C01735=-85.269,-50.626,61.037,-179.1730,-2.3238,-10409.3015
C01736=-88.593,-46.265,61.359,-179.9976,-0.1564,-10412.4256
C01737=-91.197,-41.009,61.571,179.9982,-0.0180,-10415.7877
C01738=-93.484,-35.488,61.571,179.9993,-0.0181,-10419.2124
C01739=-95.359,-29.931,61.359,179.9991,-0.1559,-10422.5741
C01740=-96.092,-24.496,61.037,179.1715,-2.3205,-10425.6986
C01741=-94.474,-19.672,60.719,176.6107,-3.5414,-10428.2376
C01742=-90.884,-16.396,60.330,172.2930,-2.2395,-10429.7735
C01743=-85.905,-15.041,59.597,172.0939,-0.5331,-10430.0688
C01744=-80.549,-13.963,58.128,174.0620,-0.3468,-10430.1656
C01745=-75.822,-12.951,56.240,177.3643,-0.2478,-10430.3070
C01746=-72.328,-11.825,54.436,-175.3679,1.0293,-10430.7148
C01747=-70.362,-9.959,53.146,-160.4056,25.5283,-10431.9439
C01748=-69.984,-6.412,52.637,-175.1539,38.4339,-10434.7651
C01749=-70.158,-3.072,52.615,179.7154,39.0245,-10437.4928
C01750=-70.224,0.000,52.630,180.0000,39.0133,-10440.0000
C01751=-70.158,3.071,52.615,-179.7148,39.0245,-10442.5064
C01752=-69.984,6.412,52.637,175.1539,38.4339,-10445.2349
C01753=-70.362,9.959,53.146,160.4106,25.5345,-10448.0561
C01754=-72.328,11.825,54.436,175.3679,1.0293,-10449.2852
C01755=-75.822,12.951,56.240,-177.3643,-0.2478,-10449.6930
C01756=-80.549,13.963,58.128,-174.0620,-0.3468,-10449.8344
C01757=-85.905,15.041,59.597,-172.0939,-0.5331,-10449.9312
C01758=-90.884,16.396,60.330,-172.2930,-2.2395,-10450.2265
C01759=-94.474,19.672,60.719,-176.6107,-3.5414,-10451.7624
C01760=-96.092,24.496,61.037,-179.1715,-2.3205,-10454.3014
C01761=-95.359,29.931,61.359,-179.9991,-0.1559,-10457.4259
C01762=-93.484,35.488,61.571,-179.9993,-0.0181,-10460.7876
C01763=-91.197,41.009,61.571,-179.9982,-0.0180,-10464.2123
C01764=-88.593,46.265,61.359,179.9976,-0.1564,-10467.5744
C01765=-85.269,50.626,61.037,179.1730,-2.3238,-10470.6985
C01766=-80.714,52.893,60.719,176.6123,-3.5381,-10473.2374
C01767=-75.858,52.671,60.330,172.2916,-2.2418,-10474.7737
C01768=-71.379,50.109,59.597,172.0924,-0.5334,-10475.0694
C01769=-66.830,47.084,58.128,174.0623,-0.3437,-10475.1660
C01770=-62.772,44.457,56.240,177.3670,-0.2495,-10475.3073
C01771=-59.505,42.782,54.436,-175.3684,1.0288,-10475.7148
C01772=-56.796,42.712,53.146,-160.4096,25.5319,-10476.9441
C01773=-54.020,44.952,52.637,-175.1533,38.4356,-10479.7651
C01774=-51.781,47.437,52.615,179.7155,39.0245,-10482.4931
C01775=-49.656,49.656,52.630,179.9948,39.0149,-10485.0000
C01776=-47.437,51.781,52.615,-179.7155,39.0245,-10487.5069
C01777=-44.952,54.020,52.637,175.1533,38.4356,-10490.2349
C01778=-42.711,56.796,53.146,160.4094,25.5317,-10493.0566
C01779=-42.782,59.505,54.436,175.3684,1.0288,-10494.2852
C01780=-44.457,62.772,56.240,-177.3670,-0.2495,-10494.6927
C01781=-47.084,66.830,58.128,-174.0623,-0.3437,-10494.8340
C01782=-50.109,71.379,59.597,-172.0924,-0.5334,-10494.9306
C01783=-52.671,75.858,60.330,-172.2916,-2.2418,-10495.2263
C01784=-52.893,80.714,60.719,-176.6123,-3.5381,-10496.7626
C01785=-50.626,85.269,61.037,-179.1730,-2.3238,-10499.3015
C01786=-46.265,88.593,61.359,-179.9976,-0.1564,-10502.4256
C01787=-41.009,91.197,61.571,179.9982,-0.0180,-10505.7877
C01788=-35.488,93.484,61.571,179.9993,-0.0181,-10509.2124
C01789=-29.931,95.359,61.359,179.9991,-0.1559,-10512.5741
C01790=-24.496,96.092,61.037,179.1715,-2.3205,-10515.6986
C01791=-19.672,94.474,60.719,176.6107,-3.5414,-10518.2376
C01792=-16.396,90.884,60.330,172.2930,-2.2395,-10519.7735
C01793=-15.041,85.905,59.597,172.0939,-0.5331,-10520.0688
C01794=-13.963,80.549,58.128,174.0620,-0.3468,-10520.1656
C01795=-12.951,75.822,56.240,177.3643,-0.2478,-10520.3070
C01796=-11.825,72.328,54.436,-175.3679,1.0293,-10520.7148
C01797=-9.959,70.362,53.146,-160.4106,25.5345,-10521.9439
C01798=-6.412,69.984,52.637,-175.1539,38.4339,-10524.7651
C01799=-3.071,70.158,52.615,179.7148,39.0245,-10527.4936
C01800=0.000,68.843,54.342,-180.0000,38.7770,-10530.0000
C01801=2.945,68.781,54.326,-179.7056,38.7871,-10532.4517
C01802=6.200,68.619,54.350,174.8933,38.1355,-10535.1629
C01803=9.699,69.044,54.888,160.3569,24.2302,-10537.9963
C01804=11.507,71.127,56.252,176.4195,0.6994,-10539.1897
C01805=12.586,74.809,58.158,-176.9112,-0.2537,-10539.5501
C01806=13.569,79.780,60.151,-173.8939,-0.2961,-10539.6525
C01807=14.621,85.405,61.698,-172.0565,-0.4508,-10539.7146
C01808=15.942,90.636,62.469,-172.2266,-2.1131,-10539.9757
C01809=19.246,94.423,62.877,-176.5198,-3.5287,-10541.5206
C01810=24.159,96.154,63.210,-179.1544,-2.3288,-10544.1038
C01811=29.718,95.429,63.547,-179.9995,-0.1559,-10547.2974
C01812=35.416,93.512,63.770,-179.9993,-0.0181,-10550.7433
C01813=41.080,91.166,63.770,-179.9982,-0.0180,-10554.2566
C01814=46.465,88.493,63.547,179.9980,-0.1564,-10557.7026
C01815=50.908,85.074,63.210,179.1554,-2.3286,-10560.8962
C01816=53.158,80.376,62.877,176.5237,-3.5316,-10563.4793
C01817=52.817,75.362,62.469,172.2314,-2.1139,-10565.0245
C01818=50.052,70.729,61.698,172.0558,-0.4490,-10565.2855
C01819=46.818,66.007,60.151,173.8890,-0.2958,-10565.3476
C01820=43.998,61.798,58.158,176.9122,-0.2494,-10565.4495
C01821=42.158,58.431,56.252,-176.4248,0.6998,-10565.8105
C01822=41.963,55.679,54.888,-160.3550,24.2338,-10567.0038
C01823=44.137,52.905,54.350,-174.8913,38.1376,-10569.8372
C01824=46.553,50.718,54.326,179.7087,38.7878,-10572.5482
C01825=48.679,48.679,54.342,179.9948,38.7763,-10575.0000
C01826=50.718,46.553,54.326,-179.7087,38.7878,-10577.4518
C01827=52.905,44.137,54.350,174.8913,38.1376,-10580.1628
C01828=55.680,41.963,54.888,160.3548,24.2336,-10582.9966
C01829=58.431,42.158,56.252,176.4248,0.6998,-10584.1895
C01830=61.798,43.998,58.158,-176.9122,-0.2494,-10584.5505
C01831=66.007,46.818,60.151,-173.8890,-0.2958,-10584.6524
C01832=70.729,50.052,61.698,-172.0558,-0.4490,-10584.7145
C01833=75.362,52.817,62.469,-172.2314,-2.1139,-10584.9755
C01834=80.376,53.158,62.877,-176.5237,-3.5316,-10586.5207
C01835=85.074,50.908,63.210,-179.1554,-2.3286,-10589.1038
C01836=88.493,46.465,63.547,-179.9980,-0.1564,-10592.2974
C01837=91.166,41.080,63.770,179.9982,-0.0180,-10595.7434
C01838=93.512,35.416,63.770,179.9993,-0.0181,-10599.2567
C01839=95.429,29.718,63.547,179.9995,-0.1559,-10602.7026
C01840=96.154,24.159,63.210,179.1544,-2.3288,-10605.8962
C01841=94.423,19.246,62.877,176.5198,-3.5287,-10608.4794
C01842=90.636,15.942,62.469,172.2266,-2.1131,-10610.0243
C01843=85.405,14.621,61.698,172.0565,-0.4508,-10610.2854
C01844=79.780,13.569,60.151,173.8939,-0.2961,-10610.3475
C01845=74.809,12.586,58.158,176.9112,-0.2537,-10610.4499
C01846=71.127,11.507,56.252,-176.4195,0.6994,-10610.8103
C01847=69.044,9.699,54.888,-160.3569,24.2302,-10612.0037
C01848=68.619,6.200,54.350,-174.8933,38.1355,-10614.8371
C01849=68.781,2.945,54.326,179.7056,38.7871,-10617.5483
C01850=68.843,0.000,54.342,-180.0000,38.7770,-10620.0000
C01851=68.781,-2.945,54.326,-179.7056,38.7871,-10622.4517
C01852=68.619,-6.200,54.350,174.8933,38.1355,-10625.1629
C01853=69.044,-9.699,54.888,160.3561,24.2357,-10627.9963
C01854=71.127,-11.507,56.252,176.4195,0.6994,-10629.1897
C01855=74.809,-12.586,58.158,-176.9112,-0.2537,-10629.5501
C01856=79.780,-13.569,60.151,-173.8939,-0.2961,-10629.6525
C01857=85.405,-14.621,61.698,-172.0565,-0.4508,-10629.7146
C01858=90.636,-15.942,62.469,-172.2266,-2.1131,-10629.9757
C01859=94.423,-19.246,62.877,-176.5198,-3.5287,-10631.5206
C01860=96.154,-24.159,63.210,-179.1544,-2.3288,-10634.1038
C01861=95.429,-29.718,63.547,-179.9995,-0.1559,-10637.2974
C01862=93.512,-35.416,63.770,-179.9993,-0.0181,-10640.7433
C01863=91.166,-41.080,63.770,-179.9982,-0.0180,-10644.2566
C01864=88.493,-46.465,63.547,179.9980,-0.1564,-10647.7026
C01865=85.074,-50.908,63.210,179.1554,-2.3286,-10650.8962
C01866=80.376,-53.158,62.877,176.5237,-3.5316,-10653.4793
C01867=75.362,-52.817,62.469,172.2314,-2.1139,-10655.0245
C01868=70.729,-50.052,61.698,172.0558,-0.4490,-10655.2855
C01869=66.007,-46.818,60.151,173.8890,-0.2958,-10655.3476
C01870=61.798,-43.998,58.158,176.9122,-0.2494,-10655.4495
C01871=58.431,-42.158,56.252,-176.4248,0.6998,-10655.8105
C01872=55.679,-41.963,54.888,-160.3550,24.2338,-10657.0038
C01873=52.905,-44.137,54.350,-174.8913,38.1376,-10659.8372
C01874=50.718,-46.553,54.326,179.7087,38.7878,-10662.5482
C01875=48.679,-48.679,54.342,179.9948,38.7763,-10665.0000
C01876=46.553,-50.718,54.326,-179.7087,38.7878,-10667.4518
C01877=44.137,-52.905,54.350,174.8913,38.1376,-10670.1628
C01878=41.963,-55.680,54.888,160.3548,24.2336,-10672.9966
C01879=42.158,-58.431,56.252,176.4248,0.6998,-10674.1895
C01880=43.998,-61.798,58.158,-176.9122,-0.2494,-10674.5505
C01881=46.818,-66.007,60.151,-173.8890,-0.2958,-10674.6524
C01882=50.052,-70.729,61.698,-172.0558,-0.4490,-10674.7145
C01883=52.817,-75.362,62.469,-172.2314,-2.1139,-10674.9755
C01884=53.158,-80.376,62.877,-176.5237,-3.5316,-10676.5207
C01885=50.908,-85.074,63.210,-179.1554,-2.3286,-10679.1038
C01886=46.465,-88.493,63.547,-179.9980,-0.1564,-10682.2974
C01887=41.080,-91.166,63.770,179.9982,-0.0180,-10685.7434
C01888=35.416,-93.512,63.770,179.9993,-0.0181,-10689.2567
C01889=29.718,-95.429,63.547,179.9995,-0.1559,-10692.7026
C01890=24.159,-96.154,63.210,179.1544,-2.3288,-10695.8962
C01891=19.246,-94.423,62.877,176.5198,-3.5287,-10698.4794
C01892=15.942,-90.636,62.469,172.2266,-2.1131,-10700.0243
C01893=14.621,-85.405,61.698,172.0565,-0.4508,-10700.2854
C01894=13.569,-79.780,60.151,173.8939,-0.2961,-10700.3475
C01895=12.586,-74.809,58.158,176.9112,-0.2537,-10700.4499
C01896=11.507,-71.127,56.252,-176.4195,0.6994,-10700.8103
C01897=9.699,-69.044,54.888,-160.3569,24.2302,-10702.0037
C01898=6.200,-68.619,54.350,-174.8933,38.1355,-10704.8371
C01899=2.945,-68.781,54.326,179.7056,38.7871,-10707.5483
C01900=0.000,-68.843,54.342,-180.0000,38.7770,-10710.0000
C01901=-2.945,-68.781,54.326,-179.7056,38.7871,-10712.4517
C01902=-6.200,-68.619,54.350,174.8933,38.1355,-10715.1629
C01903=-9.699,-69.044,54.888,160.3561,24.2357,-10717.9963
C01904=-11.507,-71.127,56.252,176.4195,0.6994,-10719.1897
C01905=-12.586,-74.809,58.158,-176.9112,-0.2537,-10719.5501
C01906=-13.569,-79.780,60.151,-173.8939,-0.2961,-10719.6525
C01907=-14.621,-85.405,61.698,-172.0565,-0.4508,-10719.7146
C01908=-15.942,-90.636,62.469,-172.2266,-2.1131,-10719.9757
C01909=-19.246,-94.423,62.877,-176.5198,-3.5287,-10721.5206
C01910=-24.159,-96.154,63.210,-179.1544,-2.3288,-10724.1038
C01911=-29.718,-95.429,63.547,-179.9995,-0.1559,-10727.2974
C01912=-35.416,-93.512,63.770,-179.9993,-0.0181,-10730.7433
C01913=-41.080,-91.166,63.770,-179.9982,-0.0180,-10734.2566
C01914=-46.465,-88.493,63.547,179.9980,-0.1564,-10737.7026
C01915=-50.908,-85.074,63.210,179.1554,-2.3286,-10740.8962
C01916=-53.158,-80.376,62.877,176.5237,-3.5316,-10743.4793
C01917=-52.817,-75.362,62.469,172.2314,-2.1139,-10745.0245
C01918=-50.052,-70.729,61.698,172.0558,-0.4490,-10745.2855
C01919=-46.818,-66.007,60.151,173.8890,-0.2958,-10745.3476
C01920=-43.998,-61.798,58.158,176.9122,-0.2494,-10745.4495
C01921=-42.158,-58.431,56.252,-176.4248,0.6998,-10745.8105
C01922=-41.963,-55.679,54.888,-160.3550,24.2338,-10747.0038
C01923=-44.137,-52.905,54.350,-174.8913,38.1376,-10749.8372
C01924=-46.553,-50.718,54.326,179.7087,38.7878,-10752.5482
C01925=-48.679,-48.679,54.342,179.9948,38.7763,-10755.0000
C01926=-50.718,-46.553,54.326,-179.7087,38.7878,-10757.4518
C01927=-52.905,-44.137,54.350,174.8913,38.1376,-10760.1628
C01928=-55.680,-41.963,54.888,160.3548,24.2336,-10762.9966
C01929=-58.431,-42.158,56.252,176.4248,0.6998,-10764.1895
C01930=-61.798,-43.998,58.158,-176.9122,-0.2494,-10764.5505
C01931=-66.007,-46.818,60.151,-173.8890,-0.2958,-10764.6524
C01932=-70.729,-50.052,61.698,-172.0558,-0.4490,-10764.7145
C01933=-75.362,-52.817,62.469,-172.2314,-2.1139,-10764.9755
C01934=-80.376,-53.158,62.877,-176.5237,-3.5316,-10766.5207
C01935=-85.074,-50.908,63.210,-179.1554,-2.3286,-10769.1038
C01936=-88.493,-46.465,63.547,-179.9980,-0.1564,-10772.2974
C01937=-91.166,-41.080,63.770,179.9982,-0.0180,-10775.7434
C01938=-93.512,-35.416,63.770,179.9993,-0.0181,-10779.2567
C01939=-95.429,-29.718,63.547,179.9995,-0.1559,-10782.7026
C01940=-96.154,-24.159,63.210,179.1544,-2.3288,-10785.8962
C01941=-94.423,-19.246,62.877,176.5198,-3.5287,-10788.4794
C01942=-90.636,-15.942,62.469,172.2266,-2.1131,-10790.0243
C01943=-85.405,-14.621,61.698,172.0565,-0.4508,-10790.2854
C01944=-79.780,-13.569,60.151,173.8939,-0.2961,-10790.3475
C01945=-74.809,-12.586,58.158,176.9112,-0.2537,-10790.4499
C01946=-71.127,-11.507,56.252,-176.4195,0.6994,-10790.8103
C01947=-69.044,-9.699,54.888,-160.3569,24.2302,-10792.0037
C01948=-68.619,-6.200,54.350,-174.8933,38.1355,-10794.8371
C01949=-68.781,-2.945,54.326,179.7056,38.7871,-10797.5483
C01950=-68.843,0.000,54.342,180.0000,38.7770,-10800.0000
C01951=-68.781,2.945,54.326,-179.7056,38.7871,-10802.4517
C01952=-68.619,6.200,54.350,174.8933,38.1355,-10805.1629
C01953=-69.044,9.699,54.888,160.3561,24.2357,-10807.9963
C01954=-71.127,11.507,56.252,176.4195,0.6994,-10809.1897
C01955=-74.809,12.586,58.158,-176.9112,-0.2537,-10809.5501
C01956=-79.780,13.569,60.151,-173.8939,-0.2961,-10809.6525
C01957=-85.405,14.621,61.698,-172.0565,-0.4508,-10809.7146
C01958=-90.636,15.942,62.469,-172.2266,-2.1131,-10809.9757
C01959=-94.423,19.246,62.877,-176.5198,-3.5287,-10811.5206
C01960=-96.154,24.159,63.210,-179.1544,-2.3288,-10814.1038
C01961=-95.429,29.718,63.547,-179.9995,-0.1559,-10817.2974
C01962=-93.512,35.416,63.770,-179.9993,-0.0181,-10820.7433
C01963=-91.166,41.080,63.770,-179.9982,-0.0180,-10824.2566
C01964=-88.493,46.465,63.547,179.9980,-0.1564,-10827.7026
C01965=-85.074,50.908,63.210,179.1554,-2.3286,-10830.8962
C01966=-80.376,53.158,62.877,176.5237,-3.5316,-10833.4793
C01967=-75.362,52.817,62.469,172.2314,-2.1139,-10835.0245
C01968=-70.729,50.052,61.698,172.0558,-0.4490,-10835.2855
C01969=-66.007,46.818,60.151,173.8890,-0.2958,-10835.3476
C01970=-61.798,43.998,58.158,176.9122,-0.2494,-10835.4495
C01971=-58.431,42.158,56.252,-176.4248,0.6998,-10835.8105
C01972=-55.679,41.963,54.888,-160.3550,24.2338,-10837.0038
C01973=-52.905,44.137,54.350,-174.8913,38.1376,-10839.8372
C01974=-50.718,46.553,54.326,179.7087,38.7878,-10842.5482
C01975=-48.679,48.679,54.342,179.9948,38.7763,-10845.0000
C01976=-46.553,50.718,54.326,-179.7087,38.7878,-10847.4518
C01977=-44.137,52.905,54.350,174.8913,38.1376,-10850.1628
C01978=-41.963,55.680,54.888,160.3548,24.2336,-10852.9966
C01979=-42.158,58.431,56.252,176.4248,0.6998,-10854.1895
C01980=-43.998,61.798,58.158,-176.9122,-0.2494,-10854.5505
C01981=-46.818,66.007,60.151,-173.8890,-0.2958,-10854.6524
C01982=-50.052,70.729,61.698,-172.0558,-0.4490,-10854.7145
C01983=-52.817,75.362,62.469,-172.2314,-2.1139,-10854.9755
C01984=-53.158,80.376,62.877,-176.5237,-3.5316,-10856.5207
C01985=-50.908,85.074,63.210,-179.1554,-2.3286,-10859.1038
C01986=-46.465,88.493,63.547,-179.9980,-0.1564,-10862.2974
C01987=-41.080,91.166,63.770,179.9982,-0.0180,-10865.7434
C01988=-35.416,93.512,63.770,179.9993,-0.0181,-10869.2567
C01989=-29.718,95.429,63.547,179.9995,-0.1559,-10872.7026
C01990=-24.159,96.154,63.210,179.1544,-2.3288,-10875.8962
C01991=-19.246,94.423,62.877,176.5198,-3.5287,-10878.4794
C01992=-15.942,90.636,62.469,172.2266,-2.1131,-10880.0243
C01993=-14.621,85.405,61.698,172.0565,-0.4508,-10880.2854
C01994=-13.569,79.780,60.151,173.8939,-0.2961,-10880.3475
C01995=-12.586,74.809,58.158,176.9112,-0.2537,-10880.4499
C01996=-11.507,71.127,56.252,-176.4195,0.6994,-10880.8103
C01997=-9.699,69.044,54.888,-160.3561,24.2357,-10882.0037
C01998=-6.200,68.619,54.350,-174.8933,38.1355,-10884.8371
C01999=-2.945,68.781,54.326,179.7056,38.7871,-10887.5483
///TOOL 0
///POSTYPE ANGLE
///ANGLE
EC00000=38.2428,7290.0000
EC00001=38.2510,7292.8792
EC00002=38.0004,7295.7259
EC00003=32.4399,7298.4654
EC00004=8.6017,7299.9566
EC00005=1.1820,7300.7254
EC00006=-0.3684,7301.2119
EC00007=-1.1362,7301.6495
EC00008=-2.4170,7302.2909
EC00009=-2.2669,7303.8024
EC00010=-1.5763,7305.9922
EC00011=-0.0779,7308.5312
EC00012=-0.0128,7311.1696
EC00013=-0.0128,7313.8303
EC00014=-0.0769,7316.4689
EC00015=-1.5754,7319.0082
EC00016=-2.2635,7321.1977
EC00017=-2.4130,7322.7089
EC00018=-1.1367,7323.3509
EC00019=-0.3687,7323.7878
EC00020=1.1799,7324.2746
EC00021=8.5989,7325.0436
EC00022=32.4425,7326.5348
EC00023=38.0014,7329.2737
EC00024=38.2519,7332.1206
EC00025=38.2429,7335.0000
EC00026=38.2519,7337.8789
EC00027=38.0014,7340.7263
EC00028=32.4425,7343.4652
EC00029=8.5989,7344.9564
EC00030=1.1799,7345.7254
EC00031=-0.3687,7346.2122
EC00032=-1.1367,7346.6491
EC00033=-2.4130,7347.2911
EC00034=-2.2635,7348.8023
EC00035=-1.5754,7350.9918
EC00036=-0.0769,7353.5311
EC00037=-0.0128,7356.1697
EC00038=-0.0128,7358.8304
EC00039=-0.0779,7361.4688
EC00040=-1.5763,7364.0078
EC00041=-2.2669,7366.1976
EC00042=-2.4170,7367.7091
EC00043=-1.1362,7368.3505
EC00044=-0.3684,7368.7881
EC00045=1.1820,7369.2746
EC00046=8.6017,7370.0434
EC00047=32.4399,7371.5346
EC00048=38.0004,7374.2741
EC00049=38.2510,7377.1208
EC00050=38.2428,7380.0000
EC00051=38.2510,7382.8792
EC00052=38.0004,7385.7266
EC00053=32.4399,7388.4654
EC00054=8.6017,7389.9566
EC00055=1.1820,7390.7254
EC00056=-0.3684,7391.2119
EC00057=-1.1362,7391.6495
EC00058=-2.4170,7392.2909
EC00059=-2.2669,7393.8024
EC00060=-1.5763,7395.9922
EC00061=-0.0779,7398.5312
EC00062=-0.0128,7401.1696
EC00063=-0.0128,7403.8303
EC00064=-0.0769,7406.4689
EC00065=-1.5754,7409.0082
EC00066=-2.2635,7411.1977
EC00067=-2.4130,7412.7089
EC00068=-1.1367,7413.3509
EC00069=-0.3687,7413.7878
EC00070=1.1799,7414.2746
EC00071=8.5989,7415.0436
EC00072=32.4425,7416.5348
EC00073=38.0014,7419.2737
EC00074=38.2519,7422.1206
EC00075=38.2429,7425.0000
EC00076=38.2519,7427.8789
EC00077=38.0014,7430.7263
EC00078=32.4425,7433.4652
EC00079=8.5989,7434.9564
EC00080=1.1799,7435.7254
EC00081=-0.3687,7436.2122
EC00082=-1.1367,7436.6491
EC00083=-2.4130,7437.2911
EC00084=-2.2635,7438.8023
EC00085=-1.5754,7440.9918
EC00086=-0.0769,7443.5311
EC00087=-0.0128,7446.1697
EC00088=-0.0128,7448.8304
EC00089=-0.0779,7451.4688
EC00090=-1.5763,7454.0078
EC00091=-2.2669,7456.1976
EC00092=-2.4170,7457.7091
EC00093=-1.1362,7458.3505
EC00094=-0.3684,7458.7881
EC00095=1.1820,7459.2746
EC00096=8.6017,7460.0434
EC00097=32.4399,7461.5346
EC00098=38.0004,7464.2741
EC00099=38.2510,7467.1208
EC00100=38.2428,7470.0000
EC00101=38.2510,7472.8792
EC00102=38.0004,7475.7266
EC00103=32.4399,7478.4654
EC00104=8.6017,7479.9566
EC00105=1.1820,7480.7254
EC00106=-0.3684,7481.2119
EC00107=-1.1362,7481.6495
EC00108=-2.4170,7482.2909
EC00109=-2.2669,7483.8024
EC00110=-1.5763,7485.9922
EC00111=-0.0779,7488.5312
EC00112=-0.0128,7491.1696
EC00113=-0.0128,7493.8303
EC00114=-0.0769,7496.4689
EC00115=-1.5754,7499.0082
EC00116=-2.2635,7501.1977
EC00117=-2.4130,7502.7089
EC00118=-1.1367,7503.3509
EC00119=-0.3687,7503.7878
EC00120=1.1799,7504.2746
EC00121=8.5989,7505.0436
EC00122=32.4425,7506.5348
EC00123=38.0014,7509.2737
EC00124=38.2519,7512.1206
EC00125=38.2429,7515.0000
EC00126=38.2519,7517.8789
EC00127=38.0014,7520.7263
EC00128=32.4425,7523.4652
EC00129=8.5989,7524.9564
EC00130=1.1799,7525.7254
EC00131=-0.3687,7526.2122
EC00132=-1.1367,7526.6491
EC00133=-2.4130,7527.2911
EC00134=-2.2635,7528.8023
EC00135=-1.5754,7530.9918
EC00136=-0.0769,7533.5311
EC00137=-0.0128,7536.1697
EC00138=-0.0128,7538.8304
EC00139=-0.0779,7541.4688
EC00140=-1.5763,7544.0078
EC00141=-2.2669,7546.1976
EC00142=-2.4170,7547.7091
EC00143=-1.1362,7548.3505
EC00144=-0.3684,7548.7881
EC00145=1.1820,7549.2746
EC00146=8.6017,7550.0434
EC00147=32.4399,7551.5346
EC00148=38.0004,7554.2741
EC00149=38.2510,7557.1208
EC00150=38.2428,7560.0000
EC00151=38.2510,7562.8792
EC00152=38.0004,7565.7266
EC00153=32.4399,7568.4654
EC00154=8.6017,7569.9566
EC00155=1.1820,7570.7254
EC00156=-0.3684,7571.2119
EC00157=-1.1362,7571.6495
EC00158=-2.4170,7572.2909
EC00159=-2.2669,7573.8024
EC00160=-1.5763,7575.9922
EC00161=-0.0779,7578.5312
EC00162=-0.0128,7581.1696
EC00163=-0.0128,7583.8303
EC00164=-0.0769,7586.4689
EC00165=-1.5754,7589.0082
EC00166=-2.2635,7591.1977
EC00167=-2.4130,7592.7089
EC00168=-1.1367,7593.3509
EC00169=-0.3687,7593.7878
EC00170=1.1799,7594.2746
EC00171=8.5989,7595.0436
EC00172=32.4425,7596.5348
EC00173=38.0014,7599.2737
EC00174=38.2519,7602.1206
EC00175=38.2429,7605.0000
EC00176=38.2519,7607.8789
EC00177=38.0014,7610.7263
EC00178=32.4425,7613.4652
EC00179=8.5989,7614.9564
EC00180=1.1799,7615.7254
EC00181=-0.3687,7616.2122
EC00182=-1.1367,7616.6491
EC00183=-2.4130,7617.2911
EC00184=-2.2635,7618.8023
EC00185=-1.5754,7620.9918
EC00186=-0.0769,7623.5311
EC00187=-0.0128,7626.1697
EC00188=-0.0128,7628.8304
EC00189=-0.0779,7631.4688
EC00190=-1.5763,7634.0078
EC00191=-2.2669,7636.1976
EC00192=-2.4170,7637.7091
EC00193=-1.1362,7638.3505
EC00194=-0.3684,7638.7881
EC00195=1.1820,7639.2746
EC00196=8.6017,7640.0434
EC00197=32.4399,7641.5346
EC00198=38.0004,7644.2734
EC00199=38.2510,7647.1208
EC00200=38.6061,7650.0000
EC00201=38.6175,7652.8388
EC00202=38.3368,7655.6728
EC00203=32.0169,7658.4202
EC00204=7.0272,7659.8823
EC00205=0.7374,7660.6084
EC00206=-0.4684,7661.0516
EC00207=-1.1309,7661.4429
EC00208=-2.5717,7662.0370
EC00209=-2.5689,7663.5473
EC00210=-1.7301,7665.7781
EC00211=-0.0960,7668.3907
EC00212=-0.0128,7671.1209
EC00213=-0.0128,7673.8793
EC00214=-0.0974,7676.6097
EC00215=-1.7292,7679.2218
EC00216=-2.5655,7681.4529
EC00217=-2.5678,7682.9628
EC00218=-1.1304,7683.5569
EC00219=-0.4635,7683.9481
EC00220=0.7386,7684.3909
EC00221=7.0239,7685.1173
EC00222=32.0179,7686.5793
EC00223=38.3333,7689.3269
EC00224=38.6195,7692.1606
EC00225=38.6039,7695.0000
EC00226=38.6195,7697.8388
EC00227=38.3333,7700.6731
EC00228=32.0179,7703.4207
EC00229=7.0239,7704.8827
EC00230=0.7386,7705.6091
EC00231=-0.4635,7706.0519
EC00232=-1.1304,7706.4431
EC00233=-2.5678,7707.0372
EC00234=-2.5655,7708.5471
EC00235=-1.7292,7710.7782
EC00236=-0.0974,7713.3903
EC00237=-0.0128,7716.1207
EC00238=-0.0128,7718.8791
EC00239=-0.0960,7721.6093
EC00240=-1.7301,7724.2219
EC00241=-2.5689,7726.4527
EC00242=-2.5717,7727.9630
EC00243=-1.1309,7728.5571
EC00244=-0.4684,7728.9484
EC00245=0.7374,7729.3916
EC00246=7.0272,7730.1177
EC00247=32.0169,7731.5798
EC00248=38.3368,7734.3272
EC00249=38.6175,7737.1612
EC00250=38.6061,7740.0000
EC00251=38.6175,7742.8388
EC00252=38.3323,7745.6728
EC00253=32.0168,7748.4209
EC00254=7.0272,7749.8823
EC00255=0.7374,7750.6084
EC00256=-0.4684,7751.0516
EC00257=-1.1309,7751.4429
EC00258=-2.5717,7752.0370
EC00259=-2.5689,7753.5473
EC00260=-1.7301,7755.7781
EC00261=-0.0960,7758.3907
EC00262=-0.0128,7761.1209
EC00263=-0.0128,7763.8793
EC00264=-0.0974,7766.6097
EC00265=-1.7292,7769.2218
EC00266=-2.5655,7771.4529
EC00267=-2.5678,7772.9628
EC00268=-1.1304,7773.5569
EC00269=-0.4635,7773.9481
EC00270=0.7386,7774.3909
EC00271=7.0239,7775.1173
EC00272=32.0179,7776.5793
EC00273=38.3333,7779.3269
EC00274=38.6195,7782.1606
EC00275=38.6039,7785.0000
EC00276=38.6195,7787.8388
EC00277=38.3333,7790.6731
EC00278=32.0179,7793.4207
EC00279=7.0239,7794.8827
EC00280=0.7386,7795.6091
EC00281=-0.4635,7796.0519
EC00282=-1.1304,7796.4431
EC00283=-2.5678,7797.0372
EC00284=-2.5655,7798.5471
EC00285=-1.7292,7800.7782
EC00286=-0.0974,7803.3903
EC00287=-0.0128,7806.1207
EC00288=-0.0128,7808.8791
EC00289=-0.0960,7811.6093
EC00290=-1.7301,7814.2219
EC00291=-2.5689,7816.4527
EC00292=-2.5717,7817.9630
EC00293=-1.1309,7818.5571
EC00294=-0.4684,7818.9484
EC00295=0.7374,7819.3916
EC00296=7.0272,7820.1177
EC00297=32.0169,7821.5798
EC00298=38.3368,7824.3272
EC00299=38.6175,7827.1612
EC00300=38.6061,7830.0000
EC00301=38.6175,7832.8388
EC00302=38.3323,7835.6728
EC00303=32.0168,7838.4209
EC00304=7.0272,7839.8823
EC00305=0.7374,7840.6084
EC00306=-0.4684,7841.0516
EC00307=-1.1309,7841.4429
EC00308=-2.5717,7842.0370
EC00309=-2.5689,7843.5473
EC00310=-1.7301,7845.7781
EC00311=-0.0960,7848.3907
EC00312=-0.0128,7851.1209
EC00313=-0.0128,7853.8793
EC00314=-0.0974,7856.6097
EC00315=-1.7292,7859.2218
EC00316=-2.5655,7861.4529
EC00317=-2.5678,7862.9628
EC00318=-1.1304,7863.5569
EC00319=-0.4635,7863.9481
EC00320=0.7386,7864.3909
EC00321=7.0239,7865.1173
EC00322=32.0179,7866.5793
EC00323=38.3333,7869.3269
EC00324=38.6195,7872.1606
EC00325=38.6039,7875.0000
EC00326=38.6195,7877.8388
EC00327=38.3333,7880.6731
EC00328=32.0179,7883.4207
EC00329=7.0239,7884.8827
EC00330=0.7386,7885.6091
EC00331=-0.4635,7886.0519
EC00332=-1.1304,7886.4431
EC00333=-2.5678,7887.0372
EC00334=-2.5655,7888.5471
EC00335=-1.7292,7890.7782
EC00336=-0.0974,7893.3903
EC00337=-0.0128,7896.1207
EC00338=-0.0128,7898.8791
EC00339=-0.0960,7901.6093
EC00340=-1.7301,7904.2219
EC00341=-2.5689,7906.4527
EC00342=-2.5717,7907.9630
EC00343=-1.1309,7908.5571
EC00344=-0.4684,7908.9484
EC00345=0.7374,7909.3916
EC00346=7.0272,7910.1177
EC00347=32.0169,7911.5798
EC00348=38.3368,7914.3272
EC00349=38.6175,7917.1612
EC00350=38.6061,7920.0000
EC00351=38.6175,7922.8388
EC00352=38.3323,7925.6728
EC00353=32.0168,7928.4209
EC00354=7.0272,7929.8823
EC00355=0.7374,7930.6084
EC00356=-0.4684,7931.0516
EC00357=-1.1309,7931.4429
EC00358=-2.5717,7932.0370
EC00359=-2.5689,7933.5473
EC00360=-1.7301,7935.7781
EC00361=-0.0960,7938.3907
EC00362=-0.0128,7941.1209
EC00363=-0.0128,7943.8793
EC00364=-0.0974,7946.6097
EC00365=-1.7292,7949.2218
EC00366=-2.5655,7951.4529
EC00367=-2.5678,7952.9628
EC00368=-1.1304,7953.5569
EC00369=-0.4635,7953.9481
EC00370=0.7386,7954.3909
EC00371=7.0239,7955.1173
EC00372=32.0179,7956.5793
EC00373=38.3333,7959.3269
EC00374=38.6195,7962.1606
EC00375=38.6039,7965.0000
EC00376=38.6195,7967.8388
EC00377=38.3333,7970.6731
EC00378=32.0179,7973.4207
EC00379=7.0239,7974.8827
EC00380=0.7386,7975.6091
EC00381=-0.4635,7976.0519
EC00382=-1.1304,7976.4431
EC00383=-2.5678,7977.0372
EC00384=-2.5655,7978.5471
EC00385=-1.7292,7980.7782
EC00386=-0.0974,7983.3903
EC00387=-0.0128,7986.1207
EC00388=-0.0128,7988.8791
EC00389=-0.0960,7991.6093
EC00390=-1.7301,7994.2219
EC00391=-2.5689,7996.4527
EC00392=-2.5717,7997.9630
EC00393=-1.1309,7998.5571
EC00394=-0.4684,7998.9484
EC00395=0.7374,7999.3916
EC00396=7.0272,8000.1177
EC00397=32.0168,8001.5791
EC00398=38.3323,8004.3272
EC00399=38.6175,8007.1612
EC00400=38.8871,8010.0000
EC00401=38.9024,8012.7966
EC00402=38.5856,8015.6177
EC00403=31.4523,8018.3745
EC00404=5.6496,8019.8055
EC00405=0.4109,8020.4884
EC00406=-0.5097,8020.8872
EC00407=-1.0814,8021.2331
EC00408=-2.6470,8021.7800
EC00409=-2.8280,8023.2896
EC00410=-1.8679,8025.5634
EC00411=-0.1087,8028.2498
EC00412=-0.0128,8031.0723
EC00413=-0.0128,8033.9275
EC00414=-0.1102,8036.7502
EC00415=-1.8680,8039.4368
EC00416=-2.8261,8041.7100
EC00417=-2.6490,8043.2198
EC00418=-1.0802,8043.7669
EC00419=-0.5117,8044.1127
EC00420=0.4096,8044.5119
EC00421=5.6466,8045.1948
EC00422=31.4493,8046.6259
EC00423=38.5888,8049.3828
EC00424=38.9007,8052.2032
EC00425=38.8857,8055.0000
EC00426=38.9007,8057.7968
EC00427=38.5853,8060.6172
EC00428=31.4493,8063.3741
EC00429=5.6466,8064.8052
EC00430=0.4096,8065.4881
EC00431=-0.5117,8065.8873
EC00432=-1.0802,8066.2331
EC00433=-2.6490,8066.7802
EC00434=-2.8261,8068.2900
EC00435=-1.8680,8070.5632
EC00436=-0.1102,8073.2498
EC00437=-0.0128,8076.0725
EC00438=-0.0128,8078.9277
EC00439=-0.1087,8081.7502
EC00440=-1.8679,8084.4366
EC00441=-2.8280,8086.7104
EC00442=-2.6470,8088.2200
EC00443=-1.0814,8088.7669
EC00444=-0.5097,8089.1128
EC00445=0.4109,8089.5116
EC00446=5.6496,8090.1945
EC00447=31.4523,8091.6255
EC00448=38.5856,8094.3823
EC00449=38.9024,8097.2034
EC00450=38.8871,8100.0000
EC00451=38.9024,8102.7966
EC00452=38.5816,8105.6177
EC00453=31.4523,8108.3745
EC00454=5.6496,8109.8055
EC00455=0.4109,8110.4884
EC00456=-0.5097,8110.8872
EC00457=-1.0814,8111.2331
EC00458=-2.6470,8111.7800
EC00459=-2.8280,8113.2896
EC00460=-1.8679,8115.5634
EC00461=-0.1087,8118.2498
EC00462=-0.0128,8121.0723
EC00463=-0.0128,8123.9275
EC00464=-0.1102,8126.7502
EC00465=-1.8680,8129.4368
EC00466=-2.8261,8131.7100
EC00467=-2.6490,8133.2198
EC00468=-1.0802,8133.7669
EC00469=-0.5117,8134.1127
EC00470=0.4096,8134.5119
EC00471=5.6466,8135.1948
EC00472=31.4493,8136.6259
EC00473=38.5888,8139.3828
EC00474=38.9007,8142.2032
EC00475=38.8857,8145.0000
EC00476=38.9007,8147.7968
EC00477=38.5853,8150.6172
EC00478=31.4493,8153.3741
EC00479=5.6466,8154.8052
EC00480=0.4096,8155.4881
EC00481=-0.5117,8155.8873
EC00482=-1.0802,8156.2331
EC00483=-2.6490,8156.7802
EC00484=-2.8261,8158.2900
EC00485=-1.8680,8160.5632
EC00486=-0.1102,8163.2498
EC00487=-0.0128,8166.0725
EC00488=-0.0128,8168.9277
EC00489=-0.1087,8171.7502
EC00490=-1.8679,8174.4366
EC00491=-2.8280,8176.7104
EC00492=-2.6470,8178.2200
EC00493=-1.0814,8178.7669
EC00494=-0.5097,8179.1128
EC00495=0.4109,8179.5116
EC00496=5.6496,8180.1945
EC00497=31.4523,8181.6255
EC00498=38.5856,8184.3823
EC00499=38.9024,8187.2034
EC00500=38.8871,8190.0000
EC00501=38.9024,8192.7966
EC00502=38.5816,8195.6177
EC00503=31.4523,8198.3745
EC00504=5.6496,8199.8055
EC00505=0.4109,8200.4884
EC00506=-0.5097,8200.8872
EC00507=-1.0814,8201.2331
EC00508=-2.6470,8201.7800
EC00509=-2.8280,8203.2896
EC00510=-1.8679,8205.5634
EC00511=-0.1087,8208.2498
EC00512=-0.0128,8211.0723
EC00513=-0.0128,8213.9275
EC00514=-0.1102,8216.7502
EC00515=-1.8680,8219.4368
EC00516=-2.8261,8221.7100
EC00517=-2.6490,8223.2198
EC00518=-1.0802,8223.7669
EC00519=-0.5117,8224.1127
EC00520=0.4096,8224.5119
EC00521=5.6466,8225.1948
EC00522=31.4493,8226.6259
EC00523=38.5888,8229.3828
EC00524=38.9007,8232.2032
EC00525=38.8857,8235.0000
EC00526=38.9007,8237.7968
EC00527=38.5853,8240.6172
EC00528=31.4493,8243.3741
EC00529=5.6466,8244.8052
EC00530=0.4096,8245.4881
EC00531=-0.5117,8245.8873
EC00532=-1.0802,8246.2331
EC00533=-2.6490,8246.7802
EC00534=-2.8261,8248.2900
EC00535=-1.8680,8250.5632
EC00536=-0.1102,8253.2498
EC00537=-0.0128,8256.0725
EC00538=-0.0128,8258.9277
EC00539=-0.1087,8261.7502
EC00540=-1.8679,8264.4366
EC00541=-2.8280,8266.7104
EC00542=-2.6470,8268.2200
EC00543=-1.0814,8268.7669
EC00544=-0.5097,8269.1128
EC00545=0.4109,8269.5116
EC00546=5.6496,8270.1945
EC00547=31.4523,8271.6255
EC00548=38.5856,8274.3823
EC00549=38.9024,8277.2034
EC00550=38.8871,8280.0000
EC00551=38.9024,8282.7966
EC00552=38.5816,8285.6177
EC00553=31.4523,8288.3745
EC00554=5.6496,8289.8055
EC00555=0.4109,8290.4884
EC00556=-0.5097,8290.8872
EC00557=-1.0814,8291.2331
EC00558=-2.6470,8291.7800
EC00559=-2.8280,8293.2896
EC00560=-1.8679,8295.5634
EC00561=-0.1087,8298.2498
EC00562=-0.0128,8301.0723
EC00563=-0.0128,8303.9275
EC00564=-0.1102,8306.7502
EC00565=-1.8680,8309.4368
EC00566=-2.8261,8311.7100
EC00567=-2.6490,8313.2198
EC00568=-1.0802,8313.7669
EC00569=-0.5117,8314.1127
EC00570=0.4096,8314.5119
EC00571=5.6466,8315.1948
EC00572=31.4493,8316.6259
EC00573=38.5888,8319.3828
EC00574=38.9007,8322.2032
EC00575=38.8857,8325.0000
EC00576=38.9007,8327.7968
EC00577=38.5853,8330.6172
EC00578=31.4493,8333.3741
EC00579=5.6466,8334.8052
EC00580=0.4096,8335.4881
EC00581=-0.5117,8335.8873
EC00582=-1.0802,8336.2331
EC00583=-2.6490,8336.7802
EC00584=-2.8261,8338.2900
EC00585=-1.8680,8340.5632
EC00586=-0.1102,8343.2498
EC00587=-0.0128,8346.0725
EC00588=-0.0128,8348.9277
EC00589=-0.1087,8351.7502
EC00590=-1.8679,8354.4366
EC00591=-2.8280,8356.7104
EC00592=-2.6470,8358.2200
EC00593=-1.0814,8358.7669
EC00594=-0.5097,8359.1128
EC00595=0.4109,8359.5116
EC00596=5.6496,8360.1945
EC00597=31.4523,8361.6255
EC00598=38.5816,8364.3823
EC00599=38.9024,8367.2034
EC00600=39.0947,8370.0000
EC00601=39.1060,8372.7531
EC00602=38.7533,8375.5598
EC00603=30.7477,8378.3257
EC00604=4.4687,8379.7254
EC00605=0.1718,8380.3637
EC00606=-0.5209,8380.7187
EC00607=-1.0036,8381.0200
EC00608=-2.6645,8381.5211
EC00609=-3.0465,8383.0317
EC00610=-1.9881,8385.3479
EC00611=-0.1196,8388.1086
EC00612=-0.0128,8391.0234
EC00613=-0.0128,8393.9765
EC00614=-0.1179,8396.8914
EC00615=-1.9866,8399.6519
EC00616=-3.0423,8401.9680
EC00617=-2.6664,8403.4791
EC00618=-1.0089,8403.9803
EC00619=-0.5237,8404.2813
EC00620=0.1687,8404.6359
EC00621=4.4679,8405.2745
EC00622=30.7469,8406.6744
EC00623=38.7545,8409.4401
EC00624=39.1054,8412.2471
EC00625=39.0946,8415.0000
EC00626=39.1054,8417.7529
EC00627=38.7545,8420.5599
EC00628=30.7510,8423.3256
EC00629=4.4679,8424.7255
EC00630=0.1687,8425.3641
EC00631=-0.5237,8425.7187
EC00632=-1.0089,8426.0197
EC00633=-2.6664,8426.5209
EC00634=-3.0423,8428.0320
EC00635=-1.9866,8430.3481
EC00636=-0.1179,8433.1086
EC00637=-0.0128,8436.0235
EC00638=-0.0128,8438.9766
EC00639=-0.1196,8441.8914
EC00640=-1.9881,8444.6521
EC00641=-3.0465,8446.9683
EC00642=-2.6645,8448.4789
EC00643=-1.0036,8448.9800
EC00644=-0.5209,8449.2813
EC00645=0.1718,8449.6363
EC00646=4.4687,8450.2746
EC00647=30.7477,8451.6743
EC00648=38.7533,8454.4402
EC00649=39.1060,8457.2469
EC00650=39.0947,8460.0000
EC00651=39.1060,8462.7531
EC00652=38.7533,8465.5598
EC00653=30.7477,8468.3257
EC00654=4.4687,8469.7254
EC00655=0.1718,8470.3637
EC00656=-0.5209,8470.7187
EC00657=-1.0036,8471.0200
EC00658=-2.6645,8471.5211
EC00659=-3.0465,8473.0317
EC00660=-1.9881,8475.3479
EC00661=-0.1196,8478.1086
EC00662=-0.0128,8481.0234
EC00663=-0.0128,8483.9765
EC00664=-0.1179,8486.8914
EC00665=-1.9866,8489.6519
EC00666=-3.0423,8491.9680
EC00667=-2.6664,8493.4791
EC00668=-1.0089,8493.9803
EC00669=-0.5237,8494.2813
EC00670=0.1687,8494.6359
EC00671=4.4679,8495.2745
EC00672=30.7469,8496.6744
EC00673=38.7545,8499.4401
EC00674=39.1054,8502.2471
EC00675=39.0946,8505.0000
EC00676=39.1054,8507.7529
EC00677=38.7545,8510.5599
EC00678=30.7510,8513.3256
EC00679=4.4679,8514.7255
EC00680=0.1687,8515.3641
EC00681=-0.5237,8515.7187
EC00682=-1.0089,8516.0197
EC00683=-2.6664,8516.5209
EC00684=-3.0423,8518.0320
EC00685=-1.9866,8520.3481
EC00686=-0.1179,8523.1086
EC00687=-0.0128,8526.0235
EC00688=-0.0128,8528.9766
EC00689=-0.1196,8531.8914
EC00690=-1.9881,8534.6521
EC00691=-3.0465,8536.9683
EC00692=-2.6645,8538.4789
EC00693=-1.0036,8538.9800
EC00694=-0.5209,8539.2813
EC00695=0.1718,8539.6363
EC00696=4.4687,8540.2746
EC00697=30.7477,8541.6743
EC00698=38.7533,8544.4402
EC00699=39.1060,8547.2469
EC00700=39.0947,8550.0000
EC00701=39.1060,8552.7531
EC00702=38.7533,8555.5598
EC00703=30.7477,8558.3257
EC00704=4.4687,8559.7254
EC00705=0.1718,8560.3637
EC00706=-0.5209,8560.7187
EC00707=-1.0036,8561.0200
EC00708=-2.6645,8561.5211
EC00709=-3.0465,8563.0317
EC00710=-1.9881,8565.3479
EC00711=-0.1196,8568.1086
EC00712=-0.0128,8571.0234
EC00713=-0.0128,8573.9765
EC00714=-0.1179,8576.8914
EC00715=-1.9866,8579.6519
EC00716=-3.0423,8581.9680
EC00717=-2.6664,8583.4791
EC00718=-1.0089,8583.9803
EC00719=-0.5237,8584.2813
EC00720=0.1687,8584.6359
EC00721=4.4679,8585.2745
EC00722=30.7469,8586.6744
EC00723=38.7545,8589.4401
EC00724=39.1054,8592.2471
EC00725=39.0946,8595.0000
EC00726=39.1054,8597.7529
EC00727=38.7545,8600.5599
EC00728=30.7510,8603.3256
EC00729=4.4679,8604.7255
EC00730=0.1687,8605.3641
EC00731=-0.5237,8605.7187
EC00732=-1.0089,8606.0197
EC00733=-2.6664,8606.5209
EC00734=-3.0423,8608.0320
EC00735=-1.9866,8610.3481
EC00736=-0.1179,8613.1086
EC00737=-0.0128,8616.0235
EC00738=-0.0128,8618.9766
EC00739=-0.1196,8621.8914
EC00740=-1.9881,8624.6521
EC00741=-3.0465,8626.9683
EC00742=-2.6645,8628.4789
EC00743=-1.0036,8628.9800
EC00744=-0.5209,8629.2813
EC00745=0.1718,8629.6363
EC00746=4.4687,8630.2746
EC00747=30.7477,8631.6743
EC00748=38.7533,8634.4402
EC00749=39.1060,8637.2469
EC00750=39.0947,8640.0000
EC00751=39.1060,8642.7531
EC00752=38.7533,8645.5598
EC00753=30.7477,8648.3257
EC00754=4.4687,8649.7254
EC00755=0.1718,8650.3637
EC00756=-0.5209,8650.7187
EC00757=-1.0036,8651.0200
EC00758=-2.6645,8651.5211
EC00759=-3.0465,8653.0317
EC00760=-1.9881,8655.3479
EC00761=-0.1196,8658.1086
EC00762=-0.0128,8661.0234
EC00763=-0.0128,8663.9765
EC00764=-0.1179,8666.8914
EC00765=-1.9866,8669.6519
EC00766=-3.0423,8671.9680
EC00767=-2.6664,8673.4791
EC00768=-1.0089,8673.9803
EC00769=-0.5237,8674.2813
EC00770=0.1687,8674.6359
EC00771=4.4679,8675.2745
EC00772=30.7469,8676.6744
EC00773=38.7545,8679.4401
EC00774=39.1054,8682.2471
EC00775=39.0946,8685.0000
EC00776=39.1054,8687.7529
EC00777=38.7545,8690.5599
EC00778=30.7510,8693.3256
EC00779=4.4679,8694.7255
EC00780=0.1687,8695.3641
EC00781=-0.5237,8695.7187
EC00782=-1.0089,8696.0197
EC00783=-2.6664,8696.5209
EC00784=-3.0423,8698.0320
EC00785=-1.9866,8700.3481
EC00786=-0.1179,8703.1086
EC00787=-0.0128,8706.0235
EC00788=-0.0128,8708.9766
EC00789=-0.1196,8711.8914
EC00790=-1.9881,8714.6521
EC00791=-3.0465,8716.9683
EC00792=-2.6645,8718.4789
EC00793=-1.0036,8718.9800
EC00794=-0.5209,8719.2813
EC00795=0.1718,8719.6363
EC00796=4.4687,8720.2746
EC00797=30.7477,8721.6743
EC00798=38.7533,8724.4402
EC00799=39.1060,8727.2469
EC00800=39.2289,8730.0000
EC00801=39.2394,8732.7075
EC00802=38.8470,8735.4993
EC00803=29.9170,8738.2758
EC00804=3.4778,8739.6431
EC00805=-0.0010,8740.2359
EC00806=-0.5058,8740.5465
EC00807=-0.9189,8740.8039
EC00808=-2.6344,8741.2607
EC00809=-3.2253,8742.7735
EC00810=-2.0919,8745.1340
EC00811=-0.1323,8747.9686
EC00812=-0.0181,8750.9753
EC00813=-0.0180,8754.0247
EC00814=-0.1307,8757.0314
EC00815=-2.0949,8759.8659
EC00816=-3.2201,8762.2261
EC00817=-2.6286,8763.7397
EC00818=-0.9152,8764.1962
EC00819=-0.5069,8764.4534
EC00820=0.0033,8764.7640
EC00821=3.4787,8765.3567
EC00822=29.9155,8766.7241
EC00823=38.8474,8769.5007
EC00824=39.2376,8772.2930
EC00825=39.2305,8775.0000
EC00826=39.2376,8777.7070
EC00827=38.8474,8780.4999
EC00828=29.9155,8783.2759
EC00829=3.4787,8784.6433
EC00830=0.0033,8785.2360
EC00831=-0.5069,8785.5466
EC00832=-0.9152,8785.8038
EC00833=-2.6286,8786.2603
EC00834=-3.2201,8787.7739
EC00835=-2.0949,8790.1341
EC00836=-0.1307,8792.9686
EC00837=-0.0180,8795.9753
EC00838=-0.0181,8799.0247
EC00839=-0.1323,8802.0314
EC00840=-2.0919,8804.8660
EC00841=-3.2253,8807.2265
EC00842=-2.6344,8808.7393
EC00843=-0.9189,8809.1961
EC00844=-0.5058,8809.4535
EC00845=-0.0010,8809.7641
EC00846=3.4778,8810.3569
EC00847=29.9170,8811.7242
EC00848=38.8470,8814.5007
EC00849=39.2394,8817.2925
EC00850=39.2289,8820.0000
EC00851=39.2394,8822.7075
EC00852=38.8470,8825.4993
EC00853=29.9170,8828.2758
EC00854=3.4778,8829.6431
EC00855=-0.0010,8830.2359
EC00856=-0.5058,8830.5465
EC00857=-0.9189,8830.8039
EC00858=-2.6344,8831.2607
EC00859=-3.2253,8832.7735
EC00860=-2.0919,8835.1340
EC00861=-0.1323,8837.9686
EC00862=-0.0181,8840.9753
EC00863=-0.0180,8844.0247
EC00864=-0.1307,8847.0314
EC00865=-2.0949,8849.8659
EC00866=-3.2201,8852.2261
EC00867=-2.6286,8853.7397
EC00868=-0.9152,8854.1962
EC00869=-0.5069,8854.4534
EC00870=0.0033,8854.7640
EC00871=3.4787,8855.3567
EC00872=29.9155,8856.7241
EC00873=38.8474,8859.5007
EC00874=39.2376,8862.2930
EC00875=39.2305,8865.0000
EC00876=39.2376,8867.7070
EC00877=38.8474,8870.4999
EC00878=29.9155,8873.2759
EC00879=3.4787,8874.6433
EC00880=0.0033,8875.2360
EC00881=-0.5069,8875.5466
EC00882=-0.9152,8875.8038
EC00883=-2.6286,8876.2603
EC00884=-3.2201,8877.7739
EC00885=-2.0949,8880.1341
EC00886=-0.1307,8882.9686
EC00887=-0.0180,8885.9753
EC00888=-0.0181,8889.0247
EC00889=-0.1323,8892.0314
EC00890=-2.0919,8894.8660
EC00891=-3.2253,8897.2265
EC00892=-2.6344,8898.7393
EC00893=-0.9189,8899.1961
EC00894=-0.5058,8899.4535
EC00895=-0.0010,8899.7641
EC00896=3.4778,8900.3569
EC00897=29.9170,8901.7242
EC00898=38.8470,8904.5007
EC00899=39.2394,8907.2925
EC00900=39.2289,8910.0000
EC00901=39.2394,8912.7075
EC00902=38.8470,8915.4993
EC00903=29.9170,8918.2758
EC00904=3.4778,8919.6431
EC00905=-0.0010,8920.2359
EC00906=-0.5058,8920.5465
EC00907=-0.9189,8920.8039
EC00908=-2.6344,8921.2607
EC00909=-3.2253,8922.7735
EC00910=-2.0919,8925.1340
EC00911=-0.1323,8927.9686
EC00912=-0.0181,8930.9753
EC00913=-0.0180,8934.0247
EC00914=-0.1307,8937.0314
EC00915=-2.0949,8939.8659
EC00916=-3.2201,8942.2261
EC00917=-2.6286,8943.7397
EC00918=-0.9152,8944.1962
EC00919=-0.5069,8944.4534
EC00920=0.0033,8944.7640
EC00921=3.4787,8945.3567
EC00922=29.9155,8946.7241
EC00923=38.8474,8949.5007
EC00924=39.2376,8952.2930
EC00925=39.2305,8955.0000
EC00926=39.2376,8957.7070
EC00927=38.8474,8960.4999
EC00928=29.9155,8963.2759
EC00929=3.4787,8964.6433
EC00930=0.0033,8965.2360
EC00931=-0.5069,8965.5466
EC00932=-0.9152,8965.8038
EC00933=-2.6286,8966.2603
EC00934=-3.2201,8967.7739
EC00935=-2.0949,8970.1341
EC00936=-0.1307,8972.9686
EC00937=-0.0180,8975.9753
EC00938=-0.0181,8979.0247
EC00939=-0.1323,8982.0314
EC00940=-2.0919,8984.8660
EC00941=-3.2253,8987.2265
EC00942=-2.6344,8988.7393
EC00943=-0.9189,8989.1961
EC00944=-0.5058,8989.4535
EC00945=-0.0010,8989.7641
EC00946=3.4778,8990.3569
EC00947=29.9170,8991.7242
EC00948=38.8470,8994.5007
EC00949=39.2394,8997.2925
EC00950=39.2289,9000.0000
EC00951=39.2394,9002.7075
EC00952=38.8470,9005.4993
EC00953=29.9170,9008.2758
EC00954=3.4778,9009.6431
EC00955=-0.0010,9010.2359
EC00956=-0.5058,9010.5465
EC00957=-0.9189,9010.8039
EC00958=-2.6344,9011.2607
EC00959=-3.2253,9012.7735
EC00960=-2.0919,9015.1340
EC00961=-0.1323,9017.9686
EC00962=-0.0181,9020.9753
EC00963=-0.0180,9024.0247
EC00964=-0.1307,9027.0314
EC00965=-2.0949,9029.8659
EC00966=-3.2201,9032.2261
EC00967=-2.6286,9033.7397
EC00968=-0.9152,9034.1962
EC00969=-0.5069,9034.4534
EC00970=0.0033,9034.7640
EC00971=3.4787,9035.3567
EC00972=29.9155,9036.7241
EC00973=38.8474,9039.5007
EC00974=39.2376,9042.2930
EC00975=39.2305,9045.0000
EC00976=39.2376,9047.7070
EC00977=38.8474,9050.4999
EC00978=29.9155,9053.2759
EC00979=3.4787,9054.6433
EC00980=0.0033,9055.2360
EC00981=-0.5069,9055.5466
EC00982=-0.9152,9055.8038
EC00983=-2.6286,9056.2603
EC00984=-3.2201,9057.7739
EC00985=-2.0949,9060.1341
EC00986=-0.1307,9062.9686
EC00987=-0.0180,9065.9753
EC00988=-0.0181,9069.0247
EC00989=-0.1323,9072.0314
EC00990=-2.0919,9074.8660
EC00991=-3.2253,9077.2265
EC00992=-2.6344,9078.7393
EC00993=-0.9189,9079.1961
EC00994=-0.5058,9079.4535
EC00995=-0.0010,9079.7641
EC00996=3.4778,9080.3569
EC00997=29.9170,9081.7242
EC00998=38.8470,9084.5007
EC00999=39.2394,9087.2925
EC01000=39.2862,9090.0000
EC01001=39.2958,9092.6603
EC01002=38.8590,9095.4368
EC01003=28.9678,9098.2235
EC01004=2.6538,9099.5577
EC01005=-0.1165,9100.1045
EC01006=-0.4746,9100.3719
EC01007=-0.8205,9100.5864
EC01008=-2.5671,9100.9998
EC01009=-3.3590,9102.5167
EC01010=-2.1798,9104.9212
EC01011=-0.1377,9107.8298
EC01012=-0.0181,9110.9268
EC01013=-0.0180,9114.0730
EC01014=-0.1358,9117.1707
EC01015=-2.1781,9120.0788
EC01016=-3.3597,9122.4830
EC01017=-2.5623,9124.0000
EC01018=-0.8206,9124.4140
EC01019=-0.4761,9124.6279
EC01020=-0.1151,9124.8952
EC01021=2.6554,9125.4421
EC01022=28.9675,9126.7764
EC01023=38.8604,9129.5628
EC01024=39.2962,9132.3404
EC01025=39.2837,9135.0000
EC01026=39.2962,9137.6596
EC01027=38.8604,9140.4372
EC01028=28.9717,9143.2236
EC01029=2.6554,9144.5579
EC01030=-0.1151,9145.1048
EC01031=-0.4761,9145.3721
EC01032=-0.8206,9145.5860
EC01033=-2.5623,9146.0000
EC01034=-3.3597,9147.5170
EC01035=-2.1781,9149.9212
EC01036=-0.1358,9152.8293
EC01037=-0.0180,9155.9270
EC01038=-0.0181,9159.0732
EC01039=-0.1377,9162.1702
EC01040=-2.1798,9165.0788
EC01041=-3.3590,9167.4833
EC01042=-2.5671,9169.0002
EC01043=-0.8205,9169.4136
EC01044=-0.4746,9169.6281
EC01045=-0.1165,9169.8955
EC01046=2.6538,9170.4423
EC01047=28.9678,9171.7765
EC01048=38.8590,9174.5632
EC01049=39.2958,9177.3397
EC01050=39.2862,9180.0000
EC01051=39.2958,9182.6603
EC01052=38.8590,9185.4368
EC01053=28.9678,9188.2235
EC01054=2.6538,9189.5577
EC01055=-0.1165,9190.1045
EC01056=-0.4746,9190.3719
EC01057=-0.8205,9190.5864
EC01058=-2.5671,9190.9998
EC01059=-3.3590,9192.5167
EC01060=-2.1798,9194.9212
EC01061=-0.1377,9197.8298
EC01062=-0.0181,9200.9268
EC01063=-0.0180,9204.0730
EC01064=-0.1358,9207.1707
EC01065=-2.1781,9210.0788
EC01066=-3.3597,9212.4830
EC01067=-2.5623,9214.0000
EC01068=-0.8206,9214.4140
EC01069=-0.4761,9214.6279
EC01070=-0.1151,9214.8952
EC01071=2.6554,9215.4421
EC01072=28.9675,9216.7764
EC01073=38.8604,9219.5628
EC01074=39.2962,9222.3404
EC01075=39.2837,9225.0000
EC01076=39.2962,9227.6596
EC01077=38.8604,9230.4372
EC01078=28.9717,9233.2236
EC01079=2.6554,9234.5579
EC01080=-0.1151,9235.1048
EC01081=-0.4761,9235.3721
EC01082=-0.8206,9235.5860
EC01083=-2.5623,9236.0000
EC01084=-3.3597,9237.5170
EC01085=-2.1781,9239.9212
EC01086=-0.1358,9242.8293
EC01087=-0.0180,9245.9270
EC01088=-0.0181,9249.0732
EC01089=-0.1377,9252.1702
EC01090=-2.1798,9255.0788
EC01091=-3.3590,9257.4833
EC01092=-2.5671,9259.0002
EC01093=-0.8205,9259.4136
EC01094=-0.4746,9259.6281
EC01095=-0.1165,9259.8955
EC01096=2.6538,9260.4423
EC01097=28.9678,9261.7765
EC01098=38.8590,9264.5632
EC01099=39.2958,9267.3397
EC01100=39.2862,9270.0000
EC01101=39.2958,9272.6603
EC01102=38.8590,9275.4368
EC01103=28.9678,9278.2235
EC01104=2.6538,9279.5577
EC01105=-0.1165,9280.1045
EC01106=-0.4746,9280.3719
EC01107=-0.8205,9280.5864
EC01108=-2.5671,9280.9998
EC01109=-3.3590,9282.5167
EC01110=-2.1798,9284.9212
EC01111=-0.1377,9287.8298
EC01112=-0.0181,9290.9268
EC01113=-0.0180,9294.0730
EC01114=-0.1358,9297.1707
EC01115=-2.1781,9300.0788
EC01116=-3.3597,9302.4830
EC01117=-2.5623,9304.0000
EC01118=-0.8206,9304.4140
EC01119=-0.4761,9304.6279
EC01120=-0.1151,9304.8952
EC01121=2.6554,9305.4421
EC01122=28.9675,9306.7764
EC01123=38.8604,9309.5628
EC01124=39.2962,9312.3404
EC01125=39.2837,9315.0000
EC01126=39.2962,9317.6596
EC01127=38.8604,9320.4372
EC01128=28.9717,9323.2236
EC01129=2.6554,9324.5579
EC01130=-0.1151,9325.1048
EC01131=-0.4761,9325.3721
EC01132=-0.8206,9325.5860
EC01133=-2.5623,9326.0000
EC01134=-3.3597,9327.5170
EC01135=-2.1781,9329.9212
EC01136=-0.1358,9332.8293
EC01137=-0.0180,9335.9270
EC01138=-0.0181,9339.0732
EC01139=-0.1377,9342.1702
EC01140=-2.1798,9345.0788
EC01141=-3.3590,9347.4833
EC01142=-2.5671,9349.0002
EC01143=-0.8205,9349.4136
EC01144=-0.4746,9349.6281
EC01145=-0.1165,9349.8955
EC01146=2.6538,9350.4423
EC01147=28.9678,9351.7765
EC01148=38.8590,9354.5632
EC01149=39.2958,9357.3397
EC01150=39.2862,9360.0000
EC01151=39.2958,9362.6603
EC01152=38.8590,9365.4368
EC01153=28.9678,9368.2235
EC01154=2.6538,9369.5577
EC01155=-0.1165,9370.1045
EC01156=-0.4746,9370.3719
EC01157=-0.8205,9370.5864
EC01158=-2.5671,9370.9998
EC01159=-3.3590,9372.5167
EC01160=-2.1798,9374.9212
EC01161=-0.1377,9377.8298
EC01162=-0.0181,9380.9268
EC01163=-0.0180,9384.0730
EC01164=-0.1358,9387.1707
EC01165=-2.1781,9390.0788
EC01166=-3.3597,9392.4830
EC01167=-2.5623,9394.0000
EC01168=-0.8206,9394.4140
EC01169=-0.4761,9394.6279
EC01170=-0.1151,9394.8952
EC01171=2.6554,9395.4421
EC01172=28.9675,9396.7764
EC01173=38.8604,9399.5628
EC01174=39.2962,9402.3404
EC01175=39.2837,9405.0000
EC01176=39.2962,9407.6596
EC01177=38.8604,9410.4372
EC01178=28.9717,9413.2236
EC01179=2.6554,9414.5579
EC01180=-0.1151,9415.1048
EC01181=-0.4761,9415.3721
EC01182=-0.8206,9415.5860
EC01183=-2.5623,9416.0000
EC01184=-3.3597,9417.5170
EC01185=-2.1781,9419.9212
EC01186=-0.1358,9422.8293
EC01187=-0.0180,9425.9270
EC01188=-0.0181,9429.0732
EC01189=-0.1377,9432.1702
EC01190=-2.1798,9435.0788
EC01191=-3.3590,9437.4833
EC01192=-2.5671,9439.0002
EC01193=-0.8205,9439.4136
EC01194=-0.4746,9439.6281
EC01195=-0.1165,9439.8955
EC01196=2.6538,9440.4423
EC01197=28.9678,9441.7765
EC01198=38.8590,9444.5632
EC01199=39.2958,9447.3397
EC01200=39.2701,9450.0000
EC01201=39.2790,9452.6105
EC01202=38.7974,9455.3720
EC01203=27.9152,9458.1701
EC01204=1.9875,9459.4699
EC01205=-0.1876,9459.9705
EC01206=-0.4381,9460.1944
EC01207=-0.7222,9460.3679
EC01208=-2.4726,9460.7398
EC01209=-3.4545,9462.2618
EC01210=-2.2474,9464.7112
EC01211=-0.1432,9467.6927
EC01212=-0.0181,9470.8797
EC01213=-0.0180,9474.1202
EC01214=-0.1435,9477.3076
EC01215=-2.2461,9480.2891
EC01216=-3.4589,9482.7379
EC01217=-2.4710,9484.2600
EC01218=-0.7206,9484.6321
EC01219=-0.4388,9484.8056
EC01220=-0.1874,9485.0300
EC01221=1.9870,9485.5299
EC01222=27.9123,9486.8301
EC01223=38.7970,9489.6279
EC01224=39.2787,9492.3891
EC01225=39.2701,9495.0000
EC01226=39.2787,9497.6109
EC01227=38.7970,9500.3721
EC01228=27.9123,9503.1699
EC01229=1.9870,9504.4701
EC01230=-0.1874,9504.9700
EC01231=-0.4388,9505.1944
EC01232=-0.7206,9505.3679
EC01233=-2.4710,9505.7400
EC01234=-3.4589,9507.2621
EC01235=-2.2461,9509.7109
EC01236=-0.1435,9512.6924
EC01237=-0.0180,9515.8798
EC01238=-0.0181,9519.1203
EC01239=-0.1432,9522.3073
EC01240=-2.2474,9525.2888
EC01241=-3.4545,9527.7382
EC01242=-2.4726,9529.2602
EC01243=-0.7222,9529.6321
EC01244=-0.4381,9529.8056
EC01245=-0.1876,9530.0295
EC01246=1.9875,9530.5301
EC01247=27.9152,9531.8299
EC01248=38.7974,9534.6280
EC01249=39.2790,9537.3895
EC01250=39.2701,9540.0000
EC01251=39.2790,9542.6105
EC01252=38.7974,9545.3720
EC01253=27.9152,9548.1701
EC01254=1.9875,9549.4699
EC01255=-0.1876,9549.9705
EC01256=-0.4381,9550.1944
EC01257=-0.7222,9550.3679
EC01258=-2.4726,9550.7398
EC01259=-3.4545,9552.2618
EC01260=-2.2474,9554.7112
EC01261=-0.1432,9557.6927
EC01262=-0.0181,9560.8797
EC01263=-0.0180,9564.1202
EC01264=-0.1435,9567.3076
EC01265=-2.2461,9570.2891
EC01266=-3.4589,9572.7379
EC01267=-2.4710,9574.2600
EC01268=-0.7206,9574.6321
EC01269=-0.4388,9574.8056
EC01270=-0.1874,9575.0300
EC01271=1.9870,9575.5299
EC01272=27.9123,9576.8301
EC01273=38.7970,9579.6279
EC01274=39.2787,9582.3891
EC01275=39.2701,9585.0000
EC01276=39.2787,9587.6109
EC01277=38.7970,9590.3721
EC01278=27.9123,9593.1699
EC01279=1.9870,9594.4701
EC01280=-0.1874,9594.9700
EC01281=-0.4388,9595.1944
EC01282=-0.7206,9595.3679
EC01283=-2.4710,9595.7400
EC01284=-3.4589,9597.2621
EC01285=-2.2461,9599.7109
EC01286=-0.1435,9602.6924
EC01287=-0.0180,9605.8798
EC01288=-0.0181,9609.1203
EC01289=-0.1432,9612.3073
EC01290=-2.2474,9615.2888
EC01291=-3.4545,9617.7382
EC01292=-2.4726,9619.2602
EC01293=-0.7222,9619.6321
EC01294=-0.4381,9619.8056
EC01295=-0.1876,9620.0295
EC01296=1.9875,9620.5301
EC01297=27.9152,9621.8299
EC01298=38.7974,9624.6280
EC01299=39.2790,9627.3895
EC01300=39.2701,9630.0000
EC01301=39.2790,9632.6105
EC01302=38.7974,9635.3720
EC01303=27.9152,9638.1701
EC01304=1.9875,9639.4699
EC01305=-0.1876,9639.9705
EC01306=-0.4381,9640.1944
EC01307=-0.7222,9640.3679
EC01308=-2.4726,9640.7398
EC01309=-3.4545,9642.2618
EC01310=-2.2474,9644.7112
EC01311=-0.1432,9647.6927
EC01312=-0.0181,9650.8797
EC01313=-0.0180,9654.1202
EC01314=-0.1435,9657.3076
EC01315=-2.2461,9660.2891
EC01316=-3.4589,9662.7379
EC01317=-2.4710,9664.2600
EC01318=-0.7206,9664.6321
EC01319=-0.4388,9664.8056
EC01320=-0.1874,9665.0300
EC01321=1.9870,9665.5299
EC01322=27.9123,9666.8301
EC01323=38.7970,9669.6279
EC01324=39.2787,9672.3891
EC01325=39.2701,9675.0000
EC01326=39.2787,9677.6109
EC01327=38.7970,9680.3721
EC01328=27.9123,9683.1699
EC01329=1.9870,9684.4701
EC01330=-0.1874,9684.9700
EC01331=-0.4388,9685.1944
EC01332=-0.7206,9685.3679
EC01333=-2.4710,9685.7400
EC01334=-3.4589,9687.2621
EC01335=-2.2461,9689.7109
EC01336=-0.1435,9692.6924
EC01337=-0.0180,9695.8798
EC01338=-0.0181,9699.1203
EC01339=-0.1432,9702.3073
EC01340=-2.2474,9705.2888
EC01341=-3.4545,9707.7382
EC01342=-2.4726,9709.2602
EC01343=-0.7222,9709.6321
EC01344=-0.4381,9709.8056
EC01345=-0.1876,9710.0295
EC01346=1.9875,9710.5301
EC01347=27.9152,9711.8299
EC01348=38.7974,9714.6280
EC01349=39.2790,9717.3895
EC01350=39.2701,9720.0000
EC01351=39.2790,9722.6105
EC01352=38.7974,9725.3720
EC01353=27.9152,9728.1701
EC01354=1.9875,9729.4699
EC01355=-0.1876,9729.9705
EC01356=-0.4381,9730.1944
EC01357=-0.7222,9730.3679
EC01358=-2.4726,9730.7398
EC01359=-3.4545,9732.2618
EC01360=-2.2474,9734.7112
EC01361=-0.1432,9737.6927
EC01362=-0.0181,9740.8797
EC01363=-0.0180,9744.1202
EC01364=-0.1435,9747.3076
EC01365=-2.2461,9750.2891
EC01366=-3.4589,9752.7379
EC01367=-2.4710,9754.2600
EC01368=-0.7206,9754.6321
EC01369=-0.4388,9754.8056
EC01370=-0.1874,9755.0300
EC01371=1.9870,9755.5299
EC01372=27.9123,9756.8301
EC01373=38.7970,9759.6279
EC01374=39.2787,9762.3891
EC01375=39.2701,9765.0000
EC01376=39.2787,9767.6109
EC01377=38.7970,9770.3721
EC01378=27.9123,9773.1699
EC01379=1.9870,9774.4701
EC01380=-0.1874,9774.9700
EC01381=-0.4388,9775.1944
EC01382=-0.7206,9775.3679
EC01383=-2.4710,9775.7400
EC01384=-3.4589,9777.2621
EC01385=-2.2461,9779.7109
EC01386=-0.1435,9782.6924
EC01387=-0.0180,9785.8798
EC01388=-0.0181,9789.1203
EC01389=-0.1432,9792.3073
EC01390=-2.2474,9795.2888
EC01391=-3.4545,9797.7382
EC01392=-2.4726,9799.2602
EC01393=-0.7222,9799.6321
EC01394=-0.4381,9799.8056
EC01395=-0.1876,9800.0295
EC01396=1.9875,9800.5301
EC01397=27.9152,9801.8299
EC01398=38.7974,9804.6280
EC01399=39.2790,9807.3895
EC01400=39.1761,9810.0000
EC01401=39.1884,9812.5595
EC01402=38.6545,9815.3045
EC01403=26.7641,9818.1135
EC01404=1.4495,9819.3788
EC01405=-0.2296,9819.8327
EC01406=-0.3936,9820.0151
EC01407=-0.6229,9820.1489
EC01408=-2.3619,9820.4816
EC01409=-3.5170,9822.0102
EC01410=-2.2970,9824.5040
EC01411=-0.1504,9827.5575
EC01412=-0.0181,9830.8329
EC01413=-0.0180,9834.1669
EC01414=-0.1486,9837.4422
EC01415=-2.2927,9840.4960
EC01416=-3.5169,9842.9901
EC01417=-2.3645,9844.5184
EC01418=-0.6241,9844.8513
EC01419=-0.3880,9844.9851
EC01420=-0.2324,9845.1672
EC01421=1.4513,9845.6212
EC01422=26.7646,9846.8860
EC01423=38.6576,9849.6950
EC01424=39.1881,9852.4397
EC01425=39.1774,9855.0000
EC01426=39.1881,9857.5591
EC01427=38.6542,9860.3050
EC01428=26.7646,9863.1140
EC01429=1.4513,9864.3788
EC01430=-0.2324,9864.8328
EC01431=-0.3880,9865.0149
EC01432=-0.6241,9865.1487
EC01433=-2.3645,9865.4816
EC01434=-3.5169,9867.0099
EC01435=-2.2927,9869.5040
EC01436=-0.1486,9872.5578
EC01437=-0.0180,9875.8331
EC01438=-0.0181,9879.1671
EC01439=-0.1504,9882.4425
EC01440=-2.2970,9885.4960
EC01441=-3.5170,9887.9898
EC01442=-2.3619,9889.5184
EC01443=-0.6229,9889.8511
EC01444=-0.3936,9889.9849
EC01445=-0.2296,9890.1673
EC01446=1.4495,9890.6212
EC01447=26.7641,9891.8865
EC01448=38.6545,9894.6955
EC01449=39.1884,9897.4405
EC01450=39.1761,9900.0000
EC01451=39.1884,9902.5595
EC01452=38.6544,9905.3053
EC01453=26.7639,9908.1143
EC01454=1.4495,9909.3788
EC01455=-0.2296,9909.8327
EC01456=-0.3936,9910.0151
EC01457=-0.6229,9910.1489
EC01458=-2.3619,9910.4816
EC01459=-3.5170,9912.0102
EC01460=-2.2970,9914.5040
EC01461=-0.1504,9917.5575
EC01462=-0.0181,9920.8329
EC01463=-0.0180,9924.1669
EC01464=-0.1486,9927.4422
EC01465=-2.2927,9930.4960
EC01466=-3.5169,9932.9901
EC01467=-2.3645,9934.5184
EC01468=-0.6241,9934.8513
EC01469=-0.3880,9934.9851
EC01470=-0.2324,9935.1672
EC01471=1.4513,9935.6212
EC01472=26.7646,9936.8860
EC01473=38.6576,9939.6950
EC01474=39.1881,9942.4397
EC01475=39.1774,9945.0000
EC01476=39.1881,9947.5591
EC01477=38.6542,9950.3050
EC01478=26.7646,9953.1140
EC01479=1.4513,9954.3788
EC01480=-0.2324,9954.8328
EC01481=-0.3880,9955.0149
EC01482=-0.6241,9955.1487
EC01483=-2.3645,9955.4816
EC01484=-3.5169,9957.0099
EC01485=-2.2927,9959.5040
EC01486=-0.1486,9962.5578
EC01487=-0.0180,9965.8331
EC01488=-0.0181,9969.1671
EC01489=-0.1504,9972.4425
EC01490=-2.2970,9975.4960
EC01491=-3.5170,9977.9898
EC01492=-2.3619,9979.5184
EC01493=-0.6229,9979.8511
EC01494=-0.3936,9979.9849
EC01495=-0.2296,9980.1673
EC01496=1.4495,9980.6212
EC01497=26.7641,9981.8865
EC01498=38.6545,9984.6955
EC01499=39.1884,9987.4405
EC01500=39.1761,9990.0000
EC01501=39.1884,9992.5595
EC01502=38.6544,9995.3053
EC01503=26.7639,9998.1143
EC01504=1.4495,9999.3788
EC01505=-0.2296,9999.8327
EC01506=-0.3936,10000.0151
EC01507=-0.6229,10000.1489
EC01508=-2.3619,10000.4816
EC01509=-3.5170,10002.0102
EC01510=-2.2970,10004.5040
EC01511=-0.1504,10007.5575
EC01512=-0.0181,10010.8329
EC01513=-0.0180,10014.1669
EC01514=-0.1486,10017.4422
EC01515=-2.2927,10020.4960
EC01516=-3.5169,10022.9901
EC01517=-2.3645,10024.5184
EC01518=-0.6241,10024.8513
EC01519=-0.3880,10024.9851
EC01520=-0.2324,10025.1672
EC01521=1.4513,10025.6212
EC01522=26.7646,10026.8860
EC01523=38.6576,10029.6950
EC01524=39.1881,10032.4397
EC01525=39.1774,10035.0000
EC01526=39.1881,10037.5591
EC01527=38.6542,10040.3050
EC01528=26.7646,10043.1140
EC01529=1.4513,10044.3788
EC01530=-0.2324,10044.8328
EC01531=-0.3880,10045.0149
EC01532=-0.6241,10045.1487
EC01533=-2.3645,10045.4816
EC01534=-3.5169,10047.0099
EC01535=-2.2927,10049.5040
EC01536=-0.1486,10052.5578
EC01537=-0.0180,10055.8331
EC01538=-0.0181,10059.1671
EC01539=-0.1504,10062.4425
EC01540=-2.2970,10065.4960
EC01541=-3.5170,10067.9898
EC01542=-2.3619,10069.5184
EC01543=-0.6229,10069.8511
EC01544=-0.3936,10069.9849
EC01545=-0.2296,10070.1673
EC01546=1.4495,10070.6212
EC01547=26.7641,10071.8865
EC01548=38.6545,10074.6955
EC01549=39.1884,10077.4405
EC01550=39.1761,10080.0000
EC01551=39.1884,10082.5595
EC01552=38.6544,10085.3053
EC01553=26.7639,10088.1143
EC01554=1.4495,10089.3788
EC01555=-0.2296,10089.8327
EC01556=-0.3936,10090.0151
EC01557=-0.6229,10090.1489
EC01558=-2.3619,10090.4816
EC01559=-3.5170,10092.0102
EC01560=-2.2970,10094.5040
EC01561=-0.1504,10097.5575
EC01562=-0.0181,10100.8329
EC01563=-0.0180,10104.1669
EC01564=-0.1486,10107.4422
EC01565=-2.2927,10110.4960
EC01566=-3.5169,10112.9901
EC01567=-2.3645,10114.5184
EC01568=-0.6241,10114.8513
EC01569=-0.3880,10114.9851
EC01570=-0.2324,10115.1672
EC01571=1.4513,10115.6212
EC01572=26.7646,10116.8860
EC01573=38.6576,10119.6950
EC01574=39.1881,10122.4397
EC01575=39.1774,10125.0000
EC01576=39.1881,10127.5591
EC01577=38.6542,10130.3050
EC01578=26.7646,10133.1140
EC01579=1.4513,10134.3788
EC01580=-0.2324,10134.8328
EC01581=-0.3880,10135.0149
EC01582=-0.6241,10135.1487
EC01583=-2.3645,10135.4816
EC01584=-3.5169,10137.0099
EC01585=-2.2927,10139.5040
EC01586=-0.1486,10142.5578
EC01587=-0.0180,10145.8331
EC01588=-0.0181,10149.1671
EC01589=-0.1504,10152.4425
EC01590=-2.2970,10155.4960
EC01591=-3.5170,10157.9898
EC01592=-2.3619,10159.5184
EC01593=-0.6229,10159.8511
EC01594=-0.3936,10159.9849
EC01595=-0.2296,10160.1673
EC01596=1.4495,10160.6212
EC01597=26.7639,10161.8857
EC01598=38.6544,10164.6947
EC01599=39.1884,10167.4405
EC01600=39.0133,10170.0000
EC01601=39.0245,10172.5072
EC01602=38.4339,10175.2349
EC01603=25.5283,10178.0561
EC01604=1.0293,10179.2852
EC01605=-0.2478,10179.6930
EC01606=-0.3468,10179.8344
EC01607=-0.5331,10179.9312
EC01608=-2.2395,10180.2265
EC01609=-3.5414,10181.7624
EC01610=-2.3205,10184.3014
EC01611=-0.1559,10187.4259
EC01612=-0.0181,10190.7876
EC01613=-0.0180,10194.2123
EC01614=-0.1564,10197.5744
EC01615=-2.3238,10200.6985
EC01616=-3.5381,10203.2374
EC01617=-2.2418,10204.7737
EC01618=-0.5334,10205.0694
EC01619=-0.3437,10205.1660
EC01620=-0.2495,10205.3073
EC01621=1.0288,10205.7148
EC01622=25.5319,10206.9441
EC01623=38.4356,10209.7651
EC01624=39.0245,10212.4931
EC01625=39.0149,10215.0000
EC01626=39.0245,10217.5069
EC01627=38.4356,10220.2349
EC01628=25.5317,10223.0566
EC01629=1.0288,10224.2852
EC01630=-0.2495,10224.6927
EC01631=-0.3437,10224.8340
EC01632=-0.5334,10224.9306
EC01633=-2.2418,10225.2263
EC01634=-3.5381,10226.7626
EC01635=-2.3238,10229.3015
EC01636=-0.1564,10232.4256
EC01637=-0.0180,10235.7877
EC01638=-0.0181,10239.2124
EC01639=-0.1559,10242.5741
EC01640=-2.3205,10245.6986
EC01641=-3.5414,10248.2376
EC01642=-2.2395,10249.7735
EC01643=-0.5331,10250.0688
EC01644=-0.3468,10250.1656
EC01645=-0.2478,10250.3070
EC01646=1.0293,10250.7148
EC01647=25.5283,10251.9439
EC01648=38.4339,10254.7651
EC01649=39.0245,10257.4928
EC01650=39.0133,10260.0000
EC01651=39.0245,10262.5064
EC01652=38.4339,10265.2349
EC01653=25.5345,10268.0561
EC01654=1.0293,10269.2852
EC01655=-0.2478,10269.6930
EC01656=-0.3468,10269.8344
EC01657=-0.5331,10269.9312
EC01658=-2.2395,10270.2265
EC01659=-3.5414,10271.7624
EC01660=-2.3205,10274.3014
EC01661=-0.1559,10277.4259
EC01662=-0.0181,10280.7876
EC01663=-0.0180,10284.2123
EC01664=-0.1564,10287.5744
EC01665=-2.3238,10290.6985
EC01666=-3.5381,10293.2374
EC01667=-2.2418,10294.7737
EC01668=-0.5334,10295.0694
EC01669=-0.3437,10295.1660
EC01670=-0.2495,10295.3073
EC01671=1.0288,10295.7148
EC01672=25.5319,10296.9441
EC01673=38.4356,10299.7651
EC01674=39.0245,10302.4931
EC01675=39.0149,10305.0000
EC01676=39.0245,10307.5069
EC01677=38.4356,10310.2349
EC01678=25.5317,10313.0566
EC01679=1.0288,10314.2852
EC01680=-0.2495,10314.6927
EC01681=-0.3437,10314.8340
EC01682=-0.5334,10314.9306
EC01683=-2.2418,10315.2263
EC01684=-3.5381,10316.7626
EC01685=-2.3238,10319.3015
EC01686=-0.1564,10322.4256
EC01687=-0.0180,10325.7877
EC01688=-0.0181,10329.2124
EC01689=-0.1559,10332.5741
EC01690=-2.3205,10335.6986
EC01691=-3.5414,10338.2376
EC01692=-2.2395,10339.7735
EC01693=-0.5331,10340.0688
EC01694=-0.3468,10340.1656
EC01695=-0.2478,10340.3070
EC01696=1.0293,10340.7148
EC01697=25.5283,10341.9439
EC01698=38.4339,10344.7651
EC01699=39.0245,10347.4928
EC01700=39.0133,10350.0000
EC01701=39.0245,10352.5064
EC01702=38.4339,10355.2349
EC01703=25.5345,10358.0561
EC01704=1.0293,10359.2852
EC01705=-0.2478,10359.6930
EC01706=-0.3468,10359.8344
EC01707=-0.5331,10359.9312
EC01708=-2.2395,10360.2265
EC01709=-3.5414,10361.7624
EC01710=-2.3205,10364.3014
EC01711=-0.1559,10367.4259
EC01712=-0.0181,10370.7876
EC01713=-0.0180,10374.2123
EC01714=-0.1564,10377.5744
EC01715=-2.3238,10380.6985
EC01716=-3.5381,10383.2374
EC01717=-2.2418,10384.7737
EC01718=-0.5334,10385.0694
EC01719=-0.3437,10385.1660
EC01720=-0.2495,10385.3073
EC01721=1.0288,10385.7148
EC01722=25.5319,10386.9441
EC01723=38.4356,10389.7651
EC01724=39.0245,10392.4931
EC01725=39.0149,10395.0000
EC01726=39.0245,10397.5069
EC01727=38.4356,10400.2349
EC01728=25.5317,10403.0566
EC01729=1.0288,10404.2852
EC01730=-0.2495,10404.6927
EC01731=-0.3437,10404.8340
EC01732=-0.5334,10404.9306
EC01733=-2.2418,10405.2263
EC01734=-3.5381,10406.7626
EC01735=-2.3238,10409.3015
EC01736=-0.1564,10412.4256
EC01737=-0.0180,10415.7877
EC01738=-0.0181,10419.2124
EC01739=-0.1559,10422.5741
EC01740=-2.3205,10425.6986
EC01741=-3.5414,10428.2376
EC01742=-2.2395,10429.7735
EC01743=-0.5331,10430.0688
EC01744=-0.3468,10430.1656
EC01745=-0.2478,10430.3070
EC01746=1.0293,10430.7148
EC01747=25.5283,10431.9439
EC01748=38.4339,10434.7651
EC01749=39.0245,10437.4928
EC01750=39.0133,10440.0000
EC01751=39.0245,10442.5064
EC01752=38.4339,10445.2349
EC01753=25.5345,10448.0561
EC01754=1.0293,10449.2852
EC01755=-0.2478,10449.6930
EC01756=-0.3468,10449.8344
EC01757=-0.5331,10449.9312
EC01758=-2.2395,10450.2265
EC01759=-3.5414,10451.7624
EC01760=-2.3205,10454.3014
EC01761=-0.1559,10457.4259
EC01762=-0.0181,10460.7876
EC01763=-0.0180,10464.2123
EC01764=-0.1564,10467.5744
EC01765=-2.3238,10470.6985
EC01766=-3.5381,10473.2374
EC01767=-2.2418,10474.7737
EC01768=-0.5334,10475.0694
EC01769=-0.3437,10475.1660
EC01770=-0.2495,10475.3073
EC01771=1.0288,10475.7148
EC01772=25.5319,10476.9441
EC01773=38.4356,10479.7651
EC01774=39.0245,10482.4931
EC01775=39.0149,10485.0000
EC01776=39.0245,10487.5069
EC01777=38.4356,10490.2349
EC01778=25.5317,10493.0566
EC01779=1.0288,10494.2852
EC01780=-0.2495,10494.6927
EC01781=-0.3437,10494.8340
EC01782=-0.5334,10494.9306
EC01783=-2.2418,10495.2263
EC01784=-3.5381,10496.7626
EC01785=-2.3238,10499.3015
EC01786=-0.1564,10502.4256
EC01787=-0.0180,10505.7877
EC01788=-0.0181,10509.2124
EC01789=-0.1559,10512.5741
EC01790=-2.3205,10515.6986
EC01791=-3.5414,10518.2376
EC01792=-2.2395,10519.7735
EC01793=-0.5331,10520.0688
EC01794=-0.3468,10520.1656
EC01795=-0.2478,10520.3070
EC01796=1.0293,10520.7148
EC01797=25.5345,10521.9439
EC01798=38.4339,10524.7651
EC01799=39.0245,10527.4936
EC01800=38.7770,10530.0000
EC01801=38.7871,10532.4517
EC01802=38.1355,10535.1629
EC01803=24.2302,10537.9963
EC01804=0.6994,10539.1897
EC01805=-0.2537,10539.5501
EC01806=-0.2961,10539.6525
EC01807=-0.4508,10539.7146
EC01808=-2.1131,10539.9757
EC01809=-3.5287,10541.5206
EC01810=-2.3288,10544.1038
EC01811=-0.1559,10547.2974
EC01812=-0.0181,10550.7433
EC01813=-0.0180,10554.2566
EC01814=-0.1564,10557.7026
EC01815=-2.3286,10560.8962
EC01816=-3.5316,10563.4793
EC01817=-2.1139,10565.0245
EC01818=-0.4490,10565.2855
EC01819=-0.2958,10565.3476
EC01820=-0.2494,10565.4495
EC01821=0.6998,10565.8105
EC01822=24.2338,10567.0038
EC01823=38.1376,10569.8372
EC01824=38.7878,10572.5482
EC01825=38.7763,10575.0000
EC01826=38.7878,10577.4518
EC01827=38.1376,10580.1628
EC01828=24.2336,10582.9966
EC01829=0.6998,10584.1895
EC01830=-0.2494,10584.5505
EC01831=-0.2958,10584.6524
EC01832=-0.4490,10584.7145
EC01833=-2.1139,10584.9755
EC01834=-3.5316,10586.5207
EC01835=-2.3286,10589.1038
EC01836=-0.1564,10592.2974
EC01837=-0.0180,10595.7434
EC01838=-0.0181,10599.2567
EC01839=-0.1559,10602.7026
EC01840=-2.3288,10605.8962
EC01841=-3.5287,10608.4794
EC01842=-2.1131,10610.0243
EC01843=-0.4508,10610.2854
EC01844=-0.2961,10610.3475
EC01845=-0.2537,10610.4499
EC01846=0.6994,10610.8103
EC01847=24.2302,10612.0037
EC01848=38.1355,10614.8371
EC01849=38.7871,10617.5483
EC01850=38.7770,10620.0000
EC01851=38.7871,10622.4517
EC01852=38.1355,10625.1629
EC01853=24.2357,10627.9963
EC01854=0.6994,10629.1897
EC01855=-0.2537,10629.5501
EC01856=-0.2961,10629.6525
EC01857=-0.4508,10629.7146
EC01858=-2.1131,10629.9757
EC01859=-3.5287,10631.5206
EC01860=-2.3288,10634.1038
EC01861=-0.1559,10637.2974
EC01862=-0.0181,10640.7433
EC01863=-0.0180,10644.2566
EC01864=-0.1564,10647.7026
EC01865=-2.3286,10650.8962
EC01866=-3.5316,10653.4793
EC01867=-2.1139,10655.0245
EC01868=-0.4490,10655.2855
EC01869=-0.2958,10655.3476
EC01870=-0.2494,10655.4495
EC01871=0.6998,10655.8105
EC01872=24.2338,10657.0038
EC01873=38.1376,10659.8372
EC01874=38.7878,10662.5482
EC01875=38.7763,10665.0000
EC01876=38.7878,10667.4518
EC01877=38.1376,10670.1628
EC01878=24.2336,10672.9966
EC01879=0.6998,10674.1895
EC01880=-0.2494,10674.5505
EC01881=-0.2958,10674.6524
EC01882=-0.4490,10674.7145
EC01883=-2.1139,10674.9755
EC01884=-3.5316,10676.5207
EC01885=-2.3286,10679.1038
EC01886=-0.1564,10682.2974
EC01887=-0.0180,10685.7434
EC01888=-0.0181,10689.2567
EC01889=-0.1559,10692.7026
EC01890=-2.3288,10695.8962
EC01891=-3.5287,10698.4794
EC01892=-2.1131,10700.0243
EC01893=-0.4508,10700.2854
EC01894=-0.2961,10700.3475
EC01895=-0.2537,10700.4499
EC01896=0.6994,10700.8103
EC01897=24.2302,10702.0037
EC01898=38.1355,10704.8371
EC01899=38.7871,10707.5483
EC01900=38.7770,10710.0000
EC01901=38.7871,10712.4517
EC01902=38.1355,10715.1629
EC01903=24.2357,10717.9963
EC01904=0.6994,10719.1897
EC01905=-0.2537,10719.5501
EC01906=-0.2961,10719.6525
EC01907=-0.4508,10719.7146
EC01908=-2.1131,10719.9757
EC01909=-3.5287,10721.5206
EC01910=-2.3288,10724.1038
EC01911=-0.1559,10727.2974
EC01912=-0.0181,10730.7433
EC01913=-0.0180,10734.2566
EC01914=-0.1564,10737.7026
EC01915=-2.3286,10740.8962
EC01916=-3.5316,10743.4793
EC01917=-2.1139,10745.0245
EC01918=-0.4490,10745.2855
EC01919=-0.2958,10745.3476
EC01920=-0.2494,10745.4495
EC01921=0.6998,10745.8105
EC01922=24.2338,10747.0038
EC01923=38.1376,10749.8372
EC01924=38.7878,10752.5482
EC01925=38.7763,10755.0000
EC01926=38.7878,10757.4518
EC01927=38.1376,10760.1628
EC01928=24.2336,10762.9966
EC01929=0.6998,10764.1895
EC01930=-0.2494,10764.5505
EC01931=-0.2958,10764.6524
EC01932=-0.4490,10764.7145
EC01933=-2.1139,10764.9755
EC01934=-3.5316,10766.5207
EC01935=-2.3286,10769.1038
EC01936=-0.1564,10772.2974
EC01937=-0.0180,10775.7434
EC01938=-0.0181,10779.2567
EC01939=-0.1559,10782.7026
EC01940=-2.3288,10785.8962
EC01941=-3.5287,10788.4794
EC01942=-2.1131,10790.0243
EC01943=-0.4508,10790.2854
EC01944=-0.2961,10790.3475
EC01945=-0.2537,10790.4499
EC01946=0.6994,10790.8103
EC01947=24.2302,10792.0037
EC01948=38.1355,10794.8371
EC01949=38.7871,10797.5483
EC01950=38.7770,10800.0000
EC01951=38.7871,10802.4517
EC01952=38.1355,10805.1629
EC01953=24.2357,10807.9963
EC01954=0.6994,10809.1897
EC01955=-0.2537,10809.5501
EC01956=-0.2961,10809.6525
EC01957=-0.4508,10809.7146
EC01958=-2.1131,10809.9757
EC01959=-3.5287,10811.5206
EC01960=-2.3288,10814.1038
EC01961=-0.1559,10817.2974
EC01962=-0.0181,10820.7433
EC01963=-0.0180,10824.2566
EC01964=-0.1564,10827.7026
EC01965=-2.3286,10830.8962
EC01966=-3.5316,10833.4793
EC01967=-2.1139,10835.0245
EC01968=-0.4490,10835.2855
EC01969=-0.2958,10835.3476
EC01970=-0.2494,10835.4495
EC01971=0.6998,10835.8105
EC01972=24.2338,10837.0038
EC01973=38.1376,10839.8372
EC01974=38.7878,10842.5482
EC01975=38.7763,10845.0000
EC01976=38.7878,10847.4518
EC01977=38.1376,10850.1628
EC01978=24.2336,10852.9966
EC01979=0.6998,10854.1895
EC01980=-0.2494,10854.5505
EC01981=-0.2958,10854.6524
EC01982=-0.4490,10854.7145
EC01983=-2.1139,10854.9755
EC01984=-3.5316,10856.5207
EC01985=-2.3286,10859.1038
EC01986=-0.1564,10862.2974
EC01987=-0.0180,10865.7434
EC01988=-0.0181,10869.2567
EC01989=-0.1559,10872.7026
EC01990=-2.3288,10875.8962
EC01991=-3.5287,10878.4794
EC01992=-2.1131,10880.0243
EC01993=-0.4508,10880.2854
EC01994=-0.2961,10880.3475
EC01995=-0.2537,10880.4499
EC01996=0.6994,10880.8103
EC01997=24.2357,10882.0037
EC01998=38.1355,10884.8371
EC01999=38.7871,10887.5483
//INST
///DATE 2021/09/24 16:41
///COMM
///ATTR SC,RW,RJ
////FRAME USER 2
///GROUP1 RB1
///GROUP2 ST1
NOP
SMOVL C00000 +MOVJ EC00000
SMOVL C00001 +MOVJ EC00001
SMOVL C00002 +MOVJ EC00002
SMOVL C00003 +MOVJ EC00003
SMOVL C00004 +MOVJ EC00004
SMOVL C00005 +MOVJ EC00005
SMOVL C00006 +MOVJ EC00006
SMOVL C00007 +MOVJ EC00007
SMOVL C00008 +MOVJ EC00008
SMOVL C00009 +MOVJ EC00009
SMOVL C00010 +MOVJ EC00010
SMOVL C00011 +MOVJ EC00011
SMOVL C00012 +MOVJ EC00012
SMOVL C00013 +MOVJ EC00013
SMOVL C00014 +MOVJ EC00014
SMOVL C00015 +MOVJ EC00015
SMOVL C00016 +MOVJ EC00016
SMOVL C00017 +MOVJ EC00017
SMOVL C00018 +MOVJ EC00018
SMOVL C00019 +MOVJ EC00019
SMOVL C00020 +MOVJ EC00020
SMOVL C00021 +MOVJ EC00021
SMOVL C00022 +MOVJ EC00022
SMOVL C00023 +MOVJ EC00023
SMOVL C00024 +MOVJ EC00024
SMOVL C00025 +MOVJ EC00025
SMOVL C00026 +MOVJ EC00026
SMOVL C00027 +MOVJ EC00027
SMOVL C00028 +MOVJ EC00028
SMOVL C00029 +MOVJ EC00029
SMOVL C00030 +MOVJ EC00030
SMOVL C00031 +MOVJ EC00031
SMOVL C00032 +MOVJ EC00032
SMOVL C00033 +MOVJ EC00033
SMOVL C00034 +MOVJ EC00034
SMOVL C00035 +MOVJ EC00035
SMOVL C00036 +MOVJ EC00036
SMOVL C00037 +MOVJ EC00037
SMOVL C00038 +MOVJ EC00038
SMOVL C00039 +MOVJ EC00039
SMOVL C00040 +MOVJ EC00040
SMOVL C00041 +MOVJ EC00041
SMOVL C00042 +MOVJ EC00042
SMOVL C00043 +MOVJ EC00043
SMOVL C00044 +MOVJ EC00044
SMOVL C00045 +MOVJ EC00045
SMOVL C00046 +MOVJ EC00046
SMOVL C00047 +MOVJ EC00047
SMOVL C00048 +MOVJ EC00048
SMOVL C00049 +MOVJ EC00049
SMOVL C00050 +MOVJ EC00050
SMOVL C00051 +MOVJ EC00051
SMOVL C00052 +MOVJ EC00052
SMOVL C00053 +MOVJ EC00053
SMOVL C00054 +MOVJ EC00054
SMOVL C00055 +MOVJ EC00055
SMOVL C00056 +MOVJ EC00056
SMOVL C00057 +MOVJ EC00057
SMOVL C00058 +MOVJ EC00058
SMOVL C00059 +MOVJ EC00059
SMOVL C00060 +MOVJ EC00060
SMOVL C00061 +MOVJ EC00061
SMOVL C00062 +MOVJ EC00062
SMOVL C00063 +MOVJ EC00063
SMOVL C00064 +MOVJ EC00064
SMOVL C00065 +MOVJ EC00065
SMOVL C00066 +MOVJ EC00066
SMOVL C00067 +MOVJ EC00067
SMOVL C00068 +MOVJ EC00068
SMOVL C00069 +MOVJ EC00069
SMOVL C00070 +MOVJ EC00070
SMOVL C00071 +MOVJ EC00071
SMOVL C00072 +MOVJ EC00072
SMOVL C00073 +MOVJ EC00073
SMOVL C00074 +MOVJ EC00074
SMOVL C00075 +MOVJ EC00075
SMOVL C00076 +MOVJ EC00076
SMOVL C00077 +MOVJ EC00077
SMOVL C00078 +MOVJ EC00078
SMOVL C00079 +MOVJ EC00079
SMOVL C00080 +MOVJ EC00080
SMOVL C00081 +MOVJ EC00081
SMOVL C00082 +MOVJ EC00082
SMOVL C00083 +MOVJ EC00083
SMOVL C00084 +MOVJ EC00084
SMOVL C00085 +MOVJ EC00085
SMOVL C00086 +MOVJ EC00086
SMOVL C00087 +MOVJ EC00087
SMOVL C00088 +MOVJ EC00088
SMOVL C00089 +MOVJ EC00089
SMOVL C00090 +MOVJ EC00090
SMOVL C00091 +MOVJ EC00091
SMOVL C00092 +MOVJ EC00092
SMOVL C00093 +MOVJ EC00093
SMOVL C00094 +MOVJ EC00094
SMOVL C00095 +MOVJ EC00095
SMOVL C00096 +MOVJ EC00096
SMOVL C00097 +MOVJ EC00097
SMOVL C00098 +MOVJ EC00098
SMOVL C00099 +MOVJ EC00099
SMOVL C00100 +MOVJ EC00100
SMOVL C00101 +MOVJ EC00101
SMOVL C00102 +MOVJ EC00102
SMOVL C00103 +MOVJ EC00103
SMOVL C00104 +MOVJ EC00104
SMOVL C00105 +MOVJ EC00105
SMOVL C00106 +MOVJ EC00106
SMOVL C00107 +MOVJ EC00107
SMOVL C00108 +MOVJ EC00108
SMOVL C00109 +MOVJ EC00109
SMOVL C00110 +MOVJ EC00110
SMOVL C00111 +MOVJ EC00111
SMOVL C00112 +MOVJ EC00112
SMOVL C00113 +MOVJ EC00113
SMOVL C00114 +MOVJ EC00114
SMOVL C00115 +MOVJ EC00115
SMOVL C00116 +MOVJ EC00116
SMOVL C00117 +MOVJ EC00117
SMOVL C00118 +MOVJ EC00118
SMOVL C00119 +MOVJ EC00119
SMOVL C00120 +MOVJ EC00120
SMOVL C00121 +MOVJ EC00121
SMOVL C00122 +MOVJ EC00122
SMOVL C00123 +MOVJ EC00123
SMOVL C00124 +MOVJ EC00124
SMOVL C00125 +MOVJ EC00125
SMOVL C00126 +MOVJ EC00126
SMOVL C00127 +MOVJ EC00127
SMOVL C00128 +MOVJ EC00128
SMOVL C00129 +MOVJ EC00129
SMOVL C00130 +MOVJ EC00130
SMOVL C00131 +MOVJ EC00131
SMOVL C00132 +MOVJ EC00132
SMOVL C00133 +MOVJ EC00133
SMOVL C00134 +MOVJ EC00134
SMOVL C00135 +MOVJ EC00135
SMOVL C00136 +MOVJ EC00136
SMOVL C00137 +MOVJ EC00137
SMOVL C00138 +MOVJ EC00138
SMOVL C00139 +MOVJ EC00139
SMOVL C00140 +MOVJ EC00140
SMOVL C00141 +MOVJ EC00141
SMOVL C00142 +MOVJ EC00142
SMOVL C00143 +MOVJ EC00143
SMOVL C00144 +MOVJ EC00144
SMOVL C00145 +MOVJ EC00145
SMOVL C00146 +MOVJ EC00146
SMOVL C00147 +MOVJ EC00147
SMOVL C00148 +MOVJ EC00148
SMOVL C00149 +MOVJ EC00149
SMOVL C00150 +MOVJ EC00150
SMOVL C00151 +MOVJ EC00151
SMOVL C00152 +MOVJ EC00152
SMOVL C00153 +MOVJ EC00153
SMOVL C00154 +MOVJ EC00154
SMOVL C00155 +MOVJ EC00155
SMOVL C00156 +MOVJ EC00156
SMOVL C00157 +MOVJ EC00157
SMOVL C00158 +MOVJ EC00158
SMOVL C00159 +MOVJ EC00159
SMOVL C00160 +MOVJ EC00160
SMOVL C00161 +MOVJ EC00161
SMOVL C00162 +MOVJ EC00162
SMOVL C00163 +MOVJ EC00163
SMOVL C00164 +MOVJ EC00164
SMOVL C00165 +MOVJ EC00165
SMOVL C00166 +MOVJ EC00166
SMOVL C00167 +MOVJ EC00167
SMOVL C00168 +MOVJ EC00168
SMOVL C00169 +MOVJ EC00169
SMOVL C00170 +MOVJ EC00170
SMOVL C00171 +MOVJ EC00171
SMOVL C00172 +MOVJ EC00172
SMOVL C00173 +MOVJ EC00173
SMOVL C00174 +MOVJ EC00174
SMOVL C00175 +MOVJ EC00175
SMOVL C00176 +MOVJ EC00176
SMOVL C00177 +MOVJ EC00177
SMOVL C00178 +MOVJ EC00178
SMOVL C00179 +MOVJ EC00179
SMOVL C00180 +MOVJ EC00180
SMOVL C00181 +MOVJ EC00181
SMOVL C00182 +MOVJ EC00182
SMOVL C00183 +MOVJ EC00183
SMOVL C00184 +MOVJ EC00184
SMOVL C00185 +MOVJ EC00185
SMOVL C00186 +MOVJ EC00186
SMOVL C00187 +MOVJ EC00187
SMOVL C00188 +MOVJ EC00188
SMOVL C00189 +MOVJ EC00189
SMOVL C00190 +MOVJ EC00190
SMOVL C00191 +MOVJ EC00191
SMOVL C00192 +MOVJ EC00192
SMOVL C00193 +MOVJ EC00193
SMOVL C00194 +MOVJ EC00194
SMOVL C00195 +MOVJ EC00195
SMOVL C00196 +MOVJ EC00196
SMOVL C00197 +MOVJ EC00197
SMOVL C00198 +MOVJ EC00198
SMOVL C00199 +MOVJ EC00199
SMOVL C00200 +MOVJ EC00200
SMOVL C00201 +MOVJ EC00201
SMOVL C00202 +MOVJ EC00202
SMOVL C00203 +MOVJ EC00203
SMOVL C00204 +MOVJ EC00204
SMOVL C00205 +MOVJ EC00205
SMOVL C00206 +MOVJ EC00206
SMOVL C00207 +MOVJ EC00207
SMOVL C00208 +MOVJ EC00208
SMOVL C00209 +MOVJ EC00209
SMOVL C00210 +MOVJ EC00210
SMOVL C00211 +MOVJ EC00211
SMOVL C00212 +MOVJ EC00212
SMOVL C00213 +MOVJ EC00213
SMOVL C00214 +MOVJ EC00214
SMOVL C00215 +MOVJ EC00215
SMOVL C00216 +MOVJ EC00216
SMOVL C00217 +MOVJ EC00217
SMOVL C00218 +MOVJ EC00218
SMOVL C00219 +MOVJ EC00219
SMOVL C00220 +MOVJ EC00220
SMOVL C00221 +MOVJ EC00221
SMOVL C00222 +MOVJ EC00222
SMOVL C00223 +MOVJ EC00223
SMOVL C00224 +MOVJ EC00224
SMOVL C00225 +MOVJ EC00225
SMOVL C00226 +MOVJ EC00226
SMOVL C00227 +MOVJ EC00227
SMOVL C00228 +MOVJ EC00228
SMOVL C00229 +MOVJ EC00229
SMOVL C00230 +MOVJ EC00230
SMOVL C00231 +MOVJ EC00231
SMOVL C00232 +MOVJ EC00232
SMOVL C00233 +MOVJ EC00233
SMOVL C00234 +MOVJ EC00234
SMOVL C00235 +MOVJ EC00235
SMOVL C00236 +MOVJ EC00236
SMOVL C00237 +MOVJ EC00237
SMOVL C00238 +MOVJ EC00238
SMOVL C00239 +MOVJ EC00239
SMOVL C00240 +MOVJ EC00240
SMOVL C00241 +MOVJ EC00241
SMOVL C00242 +MOVJ EC00242
SMOVL C00243 +MOVJ EC00243
SMOVL C00244 +MOVJ EC00244
SMOVL C00245 +MOVJ EC00245
SMOVL C00246 +MOVJ EC00246
SMOVL C00247 +MOVJ EC00247
SMOVL C00248 +MOVJ EC00248
SMOVL C00249 +MOVJ EC00249
SMOVL C00250 +MOVJ EC00250
SMOVL C00251 +MOVJ EC00251
SMOVL C00252 +MOVJ EC00252
SMOVL C00253 +MOVJ EC00253
SMOVL C00254 +MOVJ EC00254
SMOVL C00255 +MOVJ EC00255
SMOVL C00256 +MOVJ EC00256
SMOVL C00257 +MOVJ EC00257
SMOVL C00258 +MOVJ EC00258
SMOVL C00259 +MOVJ EC00259
SMOVL C00260 +MOVJ EC00260
SMOVL C00261 +MOVJ EC00261
SMOVL C00262 +MOVJ EC00262
SMOVL C00263 +MOVJ EC00263
SMOVL C00264 +MOVJ EC00264
SMOVL C00265 +MOVJ EC00265
SMOVL C00266 +MOVJ EC00266
SMOVL C00267 +MOVJ EC00267
SMOVL C00268 +MOVJ EC00268
SMOVL C00269 +MOVJ EC00269
SMOVL C00270 +MOVJ EC00270
SMOVL C00271 +MOVJ EC00271
SMOVL C00272 +MOVJ EC00272
SMOVL C00273 +MOVJ EC00273
SMOVL C00274 +MOVJ EC00274
SMOVL C00275 +MOVJ EC00275
SMOVL C00276 +MOVJ EC00276
SMOVL C00277 +MOVJ EC00277
SMOVL C00278 +MOVJ EC00278
SMOVL C00279 +MOVJ EC00279
SMOVL C00280 +MOVJ EC00280
SMOVL C00281 +MOVJ EC00281
SMOVL C00282 +MOVJ EC00282
SMOVL C00283 +MOVJ EC00283
SMOVL C00284 +MOVJ EC00284
SMOVL C00285 +MOVJ EC00285
SMOVL C00286 +MOVJ EC00286
SMOVL C00287 +MOVJ EC00287
SMOVL C00288 +MOVJ EC00288
SMOVL C00289 +MOVJ EC00289
SMOVL C00290 +MOVJ EC00290
SMOVL C00291 +MOVJ EC00291
SMOVL C00292 +MOVJ EC00292
SMOVL C00293 +MOVJ EC00293
SMOVL C00294 +MOVJ EC00294
SMOVL C00295 +MOVJ EC00295
SMOVL C00296 +MOVJ EC00296
SMOVL C00297 +MOVJ EC00297
SMOVL C00298 +MOVJ EC00298
SMOVL C00299 +MOVJ EC00299
SMOVL C00300 +MOVJ EC00300
SMOVL C00301 +MOVJ EC00301
SMOVL C00302 +MOVJ EC00302
SMOVL C00303 +MOVJ EC00303
SMOVL C00304 +MOVJ EC00304
SMOVL C00305 +MOVJ EC00305
SMOVL C00306 +MOVJ EC00306
SMOVL C00307 +MOVJ EC00307
SMOVL C00308 +MOVJ EC00308
SMOVL C00309 +MOVJ EC00309
SMOVL C00310 +MOVJ EC00310
SMOVL C00311 +MOVJ EC00311
SMOVL C00312 +MOVJ EC00312
SMOVL C00313 +MOVJ EC00313
SMOVL C00314 +MOVJ EC00314
SMOVL C00315 +MOVJ EC00315
SMOVL C00316 +MOVJ EC00316
SMOVL C00317 +MOVJ EC00317
SMOVL C00318 +MOVJ EC00318
SMOVL C00319 +MOVJ EC00319
SMOVL C00320 +MOVJ EC00320
SMOVL C00321 +MOVJ EC00321
SMOVL C00322 +MOVJ EC00322
SMOVL C00323 +MOVJ EC00323
SMOVL C00324 +MOVJ EC00324
SMOVL C00325 +MOVJ EC00325
SMOVL C00326 +MOVJ EC00326
SMOVL C00327 +MOVJ EC00327
SMOVL C00328 +MOVJ EC00328
SMOVL C00329 +MOVJ EC00329
SMOVL C00330 +MOVJ EC00330
SMOVL C00331 +MOVJ EC00331
SMOVL C00332 +MOVJ EC00332
SMOVL C00333 +MOVJ EC00333
SMOVL C00334 +MOVJ EC00334
SMOVL C00335 +MOVJ EC00335
SMOVL C00336 +MOVJ EC00336
SMOVL C00337 +MOVJ EC00337
SMOVL C00338 +MOVJ EC00338
SMOVL C00339 +MOVJ EC00339
SMOVL C00340 +MOVJ EC00340
SMOVL C00341 +MOVJ EC00341
SMOVL C00342 +MOVJ EC00342
SMOVL C00343 +MOVJ EC00343
SMOVL C00344 +MOVJ EC00344
SMOVL C00345 +MOVJ EC00345
SMOVL C00346 +MOVJ EC00346
SMOVL C00347 +MOVJ EC00347
SMOVL C00348 +MOVJ EC00348
SMOVL C00349 +MOVJ EC00349
SMOVL C00350 +MOVJ EC00350
SMOVL C00351 +MOVJ EC00351
SMOVL C00352 +MOVJ EC00352
SMOVL C00353 +MOVJ EC00353
SMOVL C00354 +MOVJ EC00354
SMOVL C00355 +MOVJ EC00355
SMOVL C00356 +MOVJ EC00356
SMOVL C00357 +MOVJ EC00357
SMOVL C00358 +MOVJ EC00358
SMOVL C00359 +MOVJ EC00359
SMOVL C00360 +MOVJ EC00360
SMOVL C00361 +MOVJ EC00361
SMOVL C00362 +MOVJ EC00362
SMOVL C00363 +MOVJ EC00363
SMOVL C00364 +MOVJ EC00364
SMOVL C00365 +MOVJ EC00365
SMOVL C00366 +MOVJ EC00366
SMOVL C00367 +MOVJ EC00367
SMOVL C00368 +MOVJ EC00368
SMOVL C00369 +MOVJ EC00369
SMOVL C00370 +MOVJ EC00370
SMOVL C00371 +MOVJ EC00371
SMOVL C00372 +MOVJ EC00372
SMOVL C00373 +MOVJ EC00373
SMOVL C00374 +MOVJ EC00374
SMOVL C00375 +MOVJ EC00375
SMOVL C00376 +MOVJ EC00376
SMOVL C00377 +MOVJ EC00377
SMOVL C00378 +MOVJ EC00378
SMOVL C00379 +MOVJ EC00379
SMOVL C00380 +MOVJ EC00380
SMOVL C00381 +MOVJ EC00381
SMOVL C00382 +MOVJ EC00382
SMOVL C00383 +MOVJ EC00383
SMOVL C00384 +MOVJ EC00384
SMOVL C00385 +MOVJ EC00385
SMOVL C00386 +MOVJ EC00386
SMOVL C00387 +MOVJ EC00387
SMOVL C00388 +MOVJ EC00388
SMOVL C00389 +MOVJ EC00389
SMOVL C00390 +MOVJ EC00390
SMOVL C00391 +MOVJ EC00391
SMOVL C00392 +MOVJ EC00392
SMOVL C00393 +MOVJ EC00393
SMOVL C00394 +MOVJ EC00394
SMOVL C00395 +MOVJ EC00395
SMOVL C00396 +MOVJ EC00396
SMOVL C00397 +MOVJ EC00397
SMOVL C00398 +MOVJ EC00398
SMOVL C00399 +MOVJ EC00399
SMOVL C00400 +MOVJ EC00400
SMOVL C00401 +MOVJ EC00401
SMOVL C00402 +MOVJ EC00402
SMOVL C00403 +MOVJ EC00403
SMOVL C00404 +MOVJ EC00404
SMOVL C00405 +MOVJ EC00405
SMOVL C00406 +MOVJ EC00406
SMOVL C00407 +MOVJ EC00407
SMOVL C00408 +MOVJ EC00408
SMOVL C00409 +MOVJ EC00409
SMOVL C00410 +MOVJ EC00410
SMOVL C00411 +MOVJ EC00411
SMOVL C00412 +MOVJ EC00412
SMOVL C00413 +MOVJ EC00413
SMOVL C00414 +MOVJ EC00414
SMOVL C00415 +MOVJ EC00415
SMOVL C00416 +MOVJ EC00416
SMOVL C00417 +MOVJ EC00417
SMOVL C00418 +MOVJ EC00418
SMOVL C00419 +MOVJ EC00419
SMOVL C00420 +MOVJ EC00420
SMOVL C00421 +MOVJ EC00421
SMOVL C00422 +MOVJ EC00422
SMOVL C00423 +MOVJ EC00423
SMOVL C00424 +MOVJ EC00424
SMOVL C00425 +MOVJ EC00425
SMOVL C00426 +MOVJ EC00426
SMOVL C00427 +MOVJ EC00427
SMOVL C00428 +MOVJ EC00428
SMOVL C00429 +MOVJ EC00429
SMOVL C00430 +MOVJ EC00430
SMOVL C00431 +MOVJ EC00431
SMOVL C00432 +MOVJ EC00432
SMOVL C00433 +MOVJ EC00433
SMOVL C00434 +MOVJ EC00434
SMOVL C00435 +MOVJ EC00435
SMOVL C00436 +MOVJ EC00436
SMOVL C00437 +MOVJ EC00437
SMOVL C00438 +MOVJ EC00438
SMOVL C00439 +MOVJ EC00439
SMOVL C00440 +MOVJ EC00440
SMOVL C00441 +MOVJ EC00441
SMOVL C00442 +MOVJ EC00442
SMOVL C00443 +MOVJ EC00443
SMOVL C00444 +MOVJ EC00444
SMOVL C00445 +MOVJ EC00445
SMOVL C00446 +MOVJ EC00446
SMOVL C00447 +MOVJ EC00447
SMOVL C00448 +MOVJ EC00448
SMOVL C00449 +MOVJ EC00449
SMOVL C00450 +MOVJ EC00450
SMOVL C00451 +MOVJ EC00451
SMOVL C00452 +MOVJ EC00452
SMOVL C00453 +MOVJ EC00453
SMOVL C00454 +MOVJ EC00454
SMOVL C00455 +MOVJ EC00455
SMOVL C00456 +MOVJ EC00456
SMOVL C00457 +MOVJ EC00457
SMOVL C00458 +MOVJ EC00458
SMOVL C00459 +MOVJ EC00459
SMOVL C00460 +MOVJ EC00460
SMOVL C00461 +MOVJ EC00461
SMOVL C00462 +MOVJ EC00462
SMOVL C00463 +MOVJ EC00463
SMOVL C00464 +MOVJ EC00464
SMOVL C00465 +MOVJ EC00465
SMOVL C00466 +MOVJ EC00466
SMOVL C00467 +MOVJ EC00467
SMOVL C00468 +MOVJ EC00468
SMOVL C00469 +MOVJ EC00469
SMOVL C00470 +MOVJ EC00470
SMOVL C00471 +MOVJ EC00471
SMOVL C00472 +MOVJ EC00472
SMOVL C00473 +MOVJ EC00473
SMOVL C00474 +MOVJ EC00474
SMOVL C00475 +MOVJ EC00475
SMOVL C00476 +MOVJ EC00476
SMOVL C00477 +MOVJ EC00477
SMOVL C00478 +MOVJ EC00478
SMOVL C00479 +MOVJ EC00479
SMOVL C00480 +MOVJ EC00480
SMOVL C00481 +MOVJ EC00481
SMOVL C00482 +MOVJ EC00482
SMOVL C00483 +MOVJ EC00483
SMOVL C00484 +MOVJ EC00484
SMOVL C00485 +MOVJ EC00485
SMOVL C00486 +MOVJ EC00486
SMOVL C00487 +MOVJ EC00487
SMOVL C00488 +MOVJ EC00488
SMOVL C00489 +MOVJ EC00489
SMOVL C00490 +MOVJ EC00490
SMOVL C00491 +MOVJ EC00491
SMOVL C00492 +MOVJ EC00492
SMOVL C00493 +MOVJ EC00493
SMOVL C00494 +MOVJ EC00494
SMOVL C00495 +MOVJ EC00495
SMOVL C00496 +MOVJ EC00496
SMOVL C00497 +MOVJ EC00497
SMOVL C00498 +MOVJ EC00498
SMOVL C00499 +MOVJ EC00499
SMOVL C00500 +MOVJ EC00500
SMOVL C00501 +MOVJ EC00501
SMOVL C00502 +MOVJ EC00502
SMOVL C00503 +MOVJ EC00503
SMOVL C00504 +MOVJ EC00504
SMOVL C00505 +MOVJ EC00505
SMOVL C00506 +MOVJ EC00506
SMOVL C00507 +MOVJ EC00507
SMOVL C00508 +MOVJ EC00508
SMOVL C00509 +MOVJ EC00509
SMOVL C00510 +MOVJ EC00510
SMOVL C00511 +MOVJ EC00511
SMOVL C00512 +MOVJ EC00512
SMOVL C00513 +MOVJ EC00513
SMOVL C00514 +MOVJ EC00514
SMOVL C00515 +MOVJ EC00515
SMOVL C00516 +MOVJ EC00516
SMOVL C00517 +MOVJ EC00517
SMOVL C00518 +MOVJ EC00518
SMOVL C00519 +MOVJ EC00519
SMOVL C00520 +MOVJ EC00520
SMOVL C00521 +MOVJ EC00521
SMOVL C00522 +MOVJ EC00522
SMOVL C00523 +MOVJ EC00523
SMOVL C00524 +MOVJ EC00524
SMOVL C00525 +MOVJ EC00525
SMOVL C00526 +MOVJ EC00526
SMOVL C00527 +MOVJ EC00527
SMOVL C00528 +MOVJ EC00528
SMOVL C00529 +MOVJ EC00529
SMOVL C00530 +MOVJ EC00530
SMOVL C00531 +MOVJ EC00531
SMOVL C00532 +MOVJ EC00532
SMOVL C00533 +MOVJ EC00533
SMOVL C00534 +MOVJ EC00534
SMOVL C00535 +MOVJ EC00535
SMOVL C00536 +MOVJ EC00536
SMOVL C00537 +MOVJ EC00537
SMOVL C00538 +MOVJ EC00538
SMOVL C00539 +MOVJ EC00539
SMOVL C00540 +MOVJ EC00540
SMOVL C00541 +MOVJ EC00541
SMOVL C00542 +MOVJ EC00542
SMOVL C00543 +MOVJ EC00543
SMOVL C00544 +MOVJ EC00544
SMOVL C00545 +MOVJ EC00545
SMOVL C00546 +MOVJ EC00546
SMOVL C00547 +MOVJ EC00547
SMOVL C00548 +MOVJ EC00548
SMOVL C00549 +MOVJ EC00549
SMOVL C00550 +MOVJ EC00550
SMOVL C00551 +MOVJ EC00551
SMOVL C00552 +MOVJ EC00552
SMOVL C00553 +MOVJ EC00553
SMOVL C00554 +MOVJ EC00554
SMOVL C00555 +MOVJ EC00555
SMOVL C00556 +MOVJ EC00556
SMOVL C00557 +MOVJ EC00557
SMOVL C00558 +MOVJ EC00558
SMOVL C00559 +MOVJ EC00559
SMOVL C00560 +MOVJ EC00560
SMOVL C00561 +MOVJ EC00561
SMOVL C00562 +MOVJ EC00562
SMOVL C00563 +MOVJ EC00563
SMOVL C00564 +MOVJ EC00564
SMOVL C00565 +MOVJ EC00565
SMOVL C00566 +MOVJ EC00566
SMOVL C00567 +MOVJ EC00567
SMOVL C00568 +MOVJ EC00568
SMOVL C00569 +MOVJ EC00569
SMOVL C00570 +MOVJ EC00570
SMOVL C00571 +MOVJ EC00571
SMOVL C00572 +MOVJ EC00572
SMOVL C00573 +MOVJ EC00573
SMOVL C00574 +MOVJ EC00574
SMOVL C00575 +MOVJ EC00575
SMOVL C00576 +MOVJ EC00576
SMOVL C00577 +MOVJ EC00577
SMOVL C00578 +MOVJ EC00578
SMOVL C00579 +MOVJ EC00579
SMOVL C00580 +MOVJ EC00580
SMOVL C00581 +MOVJ EC00581
SMOVL C00582 +MOVJ EC00582
SMOVL C00583 +MOVJ EC00583
SMOVL C00584 +MOVJ EC00584
SMOVL C00585 +MOVJ EC00585
SMOVL C00586 +MOVJ EC00586
SMOVL C00587 +MOVJ EC00587
SMOVL C00588 +MOVJ EC00588
SMOVL C00589 +MOVJ EC00589
SMOVL C00590 +MOVJ EC00590
SMOVL C00591 +MOVJ EC00591
SMOVL C00592 +MOVJ EC00592
SMOVL C00593 +MOVJ EC00593
SMOVL C00594 +MOVJ EC00594
SMOVL C00595 +MOVJ EC00595
SMOVL C00596 +MOVJ EC00596
SMOVL C00597 +MOVJ EC00597
SMOVL C00598 +MOVJ EC00598
SMOVL C00599 +MOVJ EC00599
SMOVL C00600 +MOVJ EC00600
SMOVL C00601 +MOVJ EC00601
SMOVL C00602 +MOVJ EC00602
SMOVL C00603 +MOVJ EC00603
SMOVL C00604 +MOVJ EC00604
SMOVL C00605 +MOVJ EC00605
SMOVL C00606 +MOVJ EC00606
SMOVL C00607 +MOVJ EC00607
SMOVL C00608 +MOVJ EC00608
SMOVL C00609 +MOVJ EC00609
SMOVL C00610 +MOVJ EC00610
SMOVL C00611 +MOVJ EC00611
SMOVL C00612 +MOVJ EC00612
SMOVL C00613 +MOVJ EC00613
SMOVL C00614 +MOVJ EC00614
SMOVL C00615 +MOVJ EC00615
SMOVL C00616 +MOVJ EC00616
SMOVL C00617 +MOVJ EC00617
SMOVL C00618 +MOVJ EC00618
SMOVL C00619 +MOVJ EC00619
SMOVL C00620 +MOVJ EC00620
SMOVL C00621 +MOVJ EC00621
SMOVL C00622 +MOVJ EC00622
SMOVL C00623 +MOVJ EC00623
SMOVL C00624 +MOVJ EC00624
SMOVL C00625 +MOVJ EC00625
SMOVL C00626 +MOVJ EC00626
SMOVL C00627 +MOVJ EC00627
SMOVL C00628 +MOVJ EC00628
SMOVL C00629 +MOVJ EC00629
SMOVL C00630 +MOVJ EC00630
SMOVL C00631 +MOVJ EC00631
SMOVL C00632 +MOVJ EC00632
SMOVL C00633 +MOVJ EC00633
SMOVL C00634 +MOVJ EC00634
SMOVL C00635 +MOVJ EC00635
SMOVL C00636 +MOVJ EC00636
SMOVL C00637 +MOVJ EC00637
SMOVL C00638 +MOVJ EC00638
SMOVL C00639 +MOVJ EC00639
SMOVL C00640 +MOVJ EC00640
SMOVL C00641 +MOVJ EC00641
SMOVL C00642 +MOVJ EC00642
SMOVL C00643 +MOVJ EC00643
SMOVL C00644 +MOVJ EC00644
SMOVL C00645 +MOVJ EC00645
SMOVL C00646 +MOVJ EC00646
SMOVL C00647 +MOVJ EC00647
SMOVL C00648 +MOVJ EC00648
SMOVL C00649 +MOVJ EC00649
SMOVL C00650 +MOVJ EC00650
SMOVL C00651 +MOVJ EC00651
SMOVL C00652 +MOVJ EC00652
SMOVL C00653 +MOVJ EC00653
SMOVL C00654 +MOVJ EC00654
SMOVL C00655 +MOVJ EC00655
SMOVL C00656 +MOVJ EC00656
SMOVL C00657 +MOVJ EC00657
SMOVL C00658 +MOVJ EC00658
SMOVL C00659 +MOVJ EC00659
SMOVL C00660 +MOVJ EC00660
SMOVL C00661 +MOVJ EC00661
SMOVL C00662 +MOVJ EC00662
SMOVL C00663 +MOVJ EC00663
SMOVL C00664 +MOVJ EC00664
SMOVL C00665 +MOVJ EC00665
SMOVL C00666 +MOVJ EC00666
SMOVL C00667 +MOVJ EC00667
SMOVL C00668 +MOVJ EC00668
SMOVL C00669 +MOVJ EC00669
SMOVL C00670 +MOVJ EC00670
SMOVL C00671 +MOVJ EC00671
SMOVL C00672 +MOVJ EC00672
SMOVL C00673 +MOVJ EC00673
SMOVL C00674 +MOVJ EC00674
SMOVL C00675 +MOVJ EC00675
SMOVL C00676 +MOVJ EC00676
SMOVL C00677 +MOVJ EC00677
SMOVL C00678 +MOVJ EC00678
SMOVL C00679 +MOVJ EC00679
SMOVL C00680 +MOVJ EC00680
SMOVL C00681 +MOVJ EC00681
SMOVL C00682 +MOVJ EC00682
SMOVL C00683 +MOVJ EC00683
SMOVL C00684 +MOVJ EC00684
SMOVL C00685 +MOVJ EC00685
SMOVL C00686 +MOVJ EC00686
SMOVL C00687 +MOVJ EC00687
SMOVL C00688 +MOVJ EC00688
SMOVL C00689 +MOVJ EC00689
SMOVL C00690 +MOVJ EC00690
SMOVL C00691 +MOVJ EC00691
SMOVL C00692 +MOVJ EC00692
SMOVL C00693 +MOVJ EC00693
SMOVL C00694 +MOVJ EC00694
SMOVL C00695 +MOVJ EC00695
SMOVL C00696 +MOVJ EC00696
SMOVL C00697 +MOVJ EC00697
SMOVL C00698 +MOVJ EC00698
SMOVL C00699 +MOVJ EC00699
SMOVL C00700 +MOVJ EC00700
SMOVL C00701 +MOVJ EC00701
SMOVL C00702 +MOVJ EC00702
SMOVL C00703 +MOVJ EC00703
SMOVL C00704 +MOVJ EC00704
SMOVL C00705 +MOVJ EC00705
SMOVL C00706 +MOVJ EC00706
SMOVL C00707 +MOVJ EC00707
SMOVL C00708 +MOVJ EC00708
SMOVL C00709 +MOVJ EC00709
SMOVL C00710 +MOVJ EC00710
SMOVL C00711 +MOVJ EC00711
SMOVL C00712 +MOVJ EC00712
SMOVL C00713 +MOVJ EC00713
SMOVL C00714 +MOVJ EC00714
SMOVL C00715 +MOVJ EC00715
SMOVL C00716 +MOVJ EC00716
SMOVL C00717 +MOVJ EC00717
SMOVL C00718 +MOVJ EC00718
SMOVL C00719 +MOVJ EC00719
SMOVL C00720 +MOVJ EC00720
SMOVL C00721 +MOVJ EC00721
SMOVL C00722 +MOVJ EC00722
SMOVL C00723 +MOVJ EC00723
SMOVL C00724 +MOVJ EC00724
SMOVL C00725 +MOVJ EC00725
SMOVL C00726 +MOVJ EC00726
SMOVL C00727 +MOVJ EC00727
SMOVL C00728 +MOVJ EC00728
SMOVL C00729 +MOVJ EC00729
SMOVL C00730 +MOVJ EC00730
SMOVL C00731 +MOVJ EC00731
SMOVL C00732 +MOVJ EC00732
SMOVL C00733 +MOVJ EC00733
SMOVL C00734 +MOVJ EC00734
SMOVL C00735 +MOVJ EC00735
SMOVL C00736 +MOVJ EC00736
SMOVL C00737 +MOVJ EC00737
SMOVL C00738 +MOVJ EC00738
SMOVL C00739 +MOVJ EC00739
SMOVL C00740 +MOVJ EC00740
SMOVL C00741 +MOVJ EC00741
SMOVL C00742 +MOVJ EC00742
SMOVL C00743 +MOVJ EC00743
SMOVL C00744 +MOVJ EC00744
SMOVL C00745 +MOVJ EC00745
SMOVL C00746 +MOVJ EC00746
SMOVL C00747 +MOVJ EC00747
SMOVL C00748 +MOVJ EC00748
SMOVL C00749 +MOVJ EC00749
SMOVL C00750 +MOVJ EC00750
SMOVL C00751 +MOVJ EC00751
SMOVL C00752 +MOVJ EC00752
SMOVL C00753 +MOVJ EC00753
SMOVL C00754 +MOVJ EC00754
SMOVL C00755 +MOVJ EC00755
SMOVL C00756 +MOVJ EC00756
SMOVL C00757 +MOVJ EC00757
SMOVL C00758 +MOVJ EC00758
SMOVL C00759 +MOVJ EC00759
SMOVL C00760 +MOVJ EC00760
SMOVL C00761 +MOVJ EC00761
SMOVL C00762 +MOVJ EC00762
SMOVL C00763 +MOVJ EC00763
SMOVL C00764 +MOVJ EC00764
SMOVL C00765 +MOVJ EC00765
SMOVL C00766 +MOVJ EC00766
SMOVL C00767 +MOVJ EC00767
SMOVL C00768 +MOVJ EC00768
SMOVL C00769 +MOVJ EC00769
SMOVL C00770 +MOVJ EC00770
SMOVL C00771 +MOVJ EC00771
SMOVL C00772 +MOVJ EC00772
SMOVL C00773 +MOVJ EC00773
SMOVL C00774 +MOVJ EC00774
SMOVL C00775 +MOVJ EC00775
SMOVL C00776 +MOVJ EC00776
SMOVL C00777 +MOVJ EC00777
SMOVL C00778 +MOVJ EC00778
SMOVL C00779 +MOVJ EC00779
SMOVL C00780 +MOVJ EC00780
SMOVL C00781 +MOVJ EC00781
SMOVL C00782 +MOVJ EC00782
SMOVL C00783 +MOVJ EC00783
SMOVL C00784 +MOVJ EC00784
SMOVL C00785 +MOVJ EC00785
SMOVL C00786 +MOVJ EC00786
SMOVL C00787 +MOVJ EC00787
SMOVL C00788 +MOVJ EC00788
SMOVL C00789 +MOVJ EC00789
SMOVL C00790 +MOVJ EC00790
SMOVL C00791 +MOVJ EC00791
SMOVL C00792 +MOVJ EC00792
SMOVL C00793 +MOVJ EC00793
SMOVL C00794 +MOVJ EC00794
SMOVL C00795 +MOVJ EC00795
SMOVL C00796 +MOVJ EC00796
SMOVL C00797 +MOVJ EC00797
SMOVL C00798 +MOVJ EC00798
SMOVL C00799 +MOVJ EC00799
SMOVL C00800 +MOVJ EC00800
SMOVL C00801 +MOVJ EC00801
SMOVL C00802 +MOVJ EC00802
SMOVL C00803 +MOVJ EC00803
SMOVL C00804 +MOVJ EC00804
SMOVL C00805 +MOVJ EC00805
SMOVL C00806 +MOVJ EC00806
SMOVL C00807 +MOVJ EC00807
SMOVL C00808 +MOVJ EC00808
SMOVL C00809 +MOVJ EC00809
SMOVL C00810 +MOVJ EC00810
SMOVL C00811 +MOVJ EC00811
SMOVL C00812 +MOVJ EC00812
SMOVL C00813 +MOVJ EC00813
SMOVL C00814 +MOVJ EC00814
SMOVL C00815 +MOVJ EC00815
SMOVL C00816 +MOVJ EC00816
SMOVL C00817 +MOVJ EC00817
SMOVL C00818 +MOVJ EC00818
SMOVL C00819 +MOVJ EC00819
SMOVL C00820 +MOVJ EC00820
SMOVL C00821 +MOVJ EC00821
SMOVL C00822 +MOVJ EC00822
SMOVL C00823 +MOVJ EC00823
SMOVL C00824 +MOVJ EC00824
SMOVL C00825 +MOVJ EC00825
SMOVL C00826 +MOVJ EC00826
SMOVL C00827 +MOVJ EC00827
SMOVL C00828 +MOVJ EC00828
SMOVL C00829 +MOVJ EC00829
SMOVL C00830 +MOVJ EC00830
SMOVL C00831 +MOVJ EC00831
SMOVL C00832 +MOVJ EC00832
SMOVL C00833 +MOVJ EC00833
SMOVL C00834 +MOVJ EC00834
SMOVL C00835 +MOVJ EC00835
SMOVL C00836 +MOVJ EC00836
SMOVL C00837 +MOVJ EC00837
SMOVL C00838 +MOVJ EC00838
SMOVL C00839 +MOVJ EC00839
SMOVL C00840 +MOVJ EC00840
SMOVL C00841 +MOVJ EC00841
SMOVL C00842 +MOVJ EC00842
SMOVL C00843 +MOVJ EC00843
SMOVL C00844 +MOVJ EC00844
SMOVL C00845 +MOVJ EC00845
SMOVL C00846 +MOVJ EC00846
SMOVL C00847 +MOVJ EC00847
SMOVL C00848 +MOVJ EC00848
SMOVL C00849 +MOVJ EC00849
SMOVL C00850 +MOVJ EC00850
SMOVL C00851 +MOVJ EC00851
SMOVL C00852 +MOVJ EC00852
SMOVL C00853 +MOVJ EC00853
SMOVL C00854 +MOVJ EC00854
SMOVL C00855 +MOVJ EC00855
SMOVL C00856 +MOVJ EC00856
SMOVL C00857 +MOVJ EC00857
SMOVL C00858 +MOVJ EC00858
SMOVL C00859 +MOVJ EC00859
SMOVL C00860 +MOVJ EC00860
SMOVL C00861 +MOVJ EC00861
SMOVL C00862 +MOVJ EC00862
SMOVL C00863 +MOVJ EC00863
SMOVL C00864 +MOVJ EC00864
SMOVL C00865 +MOVJ EC00865
SMOVL C00866 +MOVJ EC00866
SMOVL C00867 +MOVJ EC00867
SMOVL C00868 +MOVJ EC00868
SMOVL C00869 +MOVJ EC00869
SMOVL C00870 +MOVJ EC00870
SMOVL C00871 +MOVJ EC00871
SMOVL C00872 +MOVJ EC00872
SMOVL C00873 +MOVJ EC00873
SMOVL C00874 +MOVJ EC00874
SMOVL C00875 +MOVJ EC00875
SMOVL C00876 +MOVJ EC00876
SMOVL C00877 +MOVJ EC00877
SMOVL C00878 +MOVJ EC00878
SMOVL C00879 +MOVJ EC00879
SMOVL C00880 +MOVJ EC00880
SMOVL C00881 +MOVJ EC00881
SMOVL C00882 +MOVJ EC00882
SMOVL C00883 +MOVJ EC00883
SMOVL C00884 +MOVJ EC00884
SMOVL C00885 +MOVJ EC00885
SMOVL C00886 +MOVJ EC00886
SMOVL C00887 +MOVJ EC00887
SMOVL C00888 +MOVJ EC00888
SMOVL C00889 +MOVJ EC00889
SMOVL C00890 +MOVJ EC00890
SMOVL C00891 +MOVJ EC00891
SMOVL C00892 +MOVJ EC00892
SMOVL C00893 +MOVJ EC00893
SMOVL C00894 +MOVJ EC00894
SMOVL C00895 +MOVJ EC00895
SMOVL C00896 +MOVJ EC00896
SMOVL C00897 +MOVJ EC00897
SMOVL C00898 +MOVJ EC00898
SMOVL C00899 +MOVJ EC00899
SMOVL C00900 +MOVJ EC00900
SMOVL C00901 +MOVJ EC00901
SMOVL C00902 +MOVJ EC00902
SMOVL C00903 +MOVJ EC00903
SMOVL C00904 +MOVJ EC00904
SMOVL C00905 +MOVJ EC00905
SMOVL C00906 +MOVJ EC00906
SMOVL C00907 +MOVJ EC00907
SMOVL C00908 +MOVJ EC00908
SMOVL C00909 +MOVJ EC00909
SMOVL C00910 +MOVJ EC00910
SMOVL C00911 +MOVJ EC00911
SMOVL C00912 +MOVJ EC00912
SMOVL C00913 +MOVJ EC00913
SMOVL C00914 +MOVJ EC00914
SMOVL C00915 +MOVJ EC00915
SMOVL C00916 +MOVJ EC00916
SMOVL C00917 +MOVJ EC00917
SMOVL C00918 +MOVJ EC00918
SMOVL C00919 +MOVJ EC00919
SMOVL C00920 +MOVJ EC00920
SMOVL C00921 +MOVJ EC00921
SMOVL C00922 +MOVJ EC00922
SMOVL C00923 +MOVJ EC00923
SMOVL C00924 +MOVJ EC00924
SMOVL C00925 +MOVJ EC00925
SMOVL C00926 +MOVJ EC00926
SMOVL C00927 +MOVJ EC00927
SMOVL C00928 +MOVJ EC00928
SMOVL C00929 +MOVJ EC00929
SMOVL C00930 +MOVJ EC00930
SMOVL C00931 +MOVJ EC00931
SMOVL C00932 +MOVJ EC00932
SMOVL C00933 +MOVJ EC00933
SMOVL C00934 +MOVJ EC00934
SMOVL C00935 +MOVJ EC00935
SMOVL C00936 +MOVJ EC00936
SMOVL C00937 +MOVJ EC00937
SMOVL C00938 +MOVJ EC00938
SMOVL C00939 +MOVJ EC00939
SMOVL C00940 +MOVJ EC00940
SMOVL C00941 +MOVJ EC00941
SMOVL C00942 +MOVJ EC00942
SMOVL C00943 +MOVJ EC00943
SMOVL C00944 +MOVJ EC00944
SMOVL C00945 +MOVJ EC00945
SMOVL C00946 +MOVJ EC00946
SMOVL C00947 +MOVJ EC00947
SMOVL C00948 +MOVJ EC00948
SMOVL C00949 +MOVJ EC00949
SMOVL C00950 +MOVJ EC00950
SMOVL C00951 +MOVJ EC00951
SMOVL C00952 +MOVJ EC00952
SMOVL C00953 +MOVJ EC00953
SMOVL C00954 +MOVJ EC00954
SMOVL C00955 +MOVJ EC00955
SMOVL C00956 +MOVJ EC00956
SMOVL C00957 +MOVJ EC00957
SMOVL C00958 +MOVJ EC00958
SMOVL C00959 +MOVJ EC00959
SMOVL C00960 +MOVJ EC00960
SMOVL C00961 +MOVJ EC00961
SMOVL C00962 +MOVJ EC00962
SMOVL C00963 +MOVJ EC00963
SMOVL C00964 +MOVJ EC00964
SMOVL C00965 +MOVJ EC00965
SMOVL C00966 +MOVJ EC00966
SMOVL C00967 +MOVJ EC00967
SMOVL C00968 +MOVJ EC00968
SMOVL C00969 +MOVJ EC00969
SMOVL C00970 +MOVJ EC00970
SMOVL C00971 +MOVJ EC00971
SMOVL C00972 +MOVJ EC00972
SMOVL C00973 +MOVJ EC00973
SMOVL C00974 +MOVJ EC00974
SMOVL C00975 +MOVJ EC00975
SMOVL C00976 +MOVJ EC00976
SMOVL C00977 +MOVJ EC00977
SMOVL C00978 +MOVJ EC00978
SMOVL C00979 +MOVJ EC00979
SMOVL C00980 +MOVJ EC00980
SMOVL C00981 +MOVJ EC00981
SMOVL C00982 +MOVJ EC00982
SMOVL C00983 +MOVJ EC00983
SMOVL C00984 +MOVJ EC00984
SMOVL C00985 +MOVJ EC00985
SMOVL C00986 +MOVJ EC00986
SMOVL C00987 +MOVJ EC00987
SMOVL C00988 +MOVJ EC00988
SMOVL C00989 +MOVJ EC00989
SMOVL C00990 +MOVJ EC00990
SMOVL C00991 +MOVJ EC00991
SMOVL C00992 +MOVJ EC00992
SMOVL C00993 +MOVJ EC00993
SMOVL C00994 +MOVJ EC00994
SMOVL C00995 +MOVJ EC00995
SMOVL C00996 +MOVJ EC00996
SMOVL C00997 +MOVJ EC00997
SMOVL C00998 +MOVJ EC00998
SMOVL C00999 +MOVJ EC00999
SMOVL C01000 +MOVJ EC01000
SMOVL C01001 +MOVJ EC01001
SMOVL C01002 +MOVJ EC01002
SMOVL C01003 +MOVJ EC01003
SMOVL C01004 +MOVJ EC01004
SMOVL C01005 +MOVJ EC01005
SMOVL C01006 +MOVJ EC01006
SMOVL C01007 +MOVJ EC01007
SMOVL C01008 +MOVJ EC01008
SMOVL C01009 +MOVJ EC01009
SMOVL C01010 +MOVJ EC01010
SMOVL C01011 +MOVJ EC01011
SMOVL C01012 +MOVJ EC01012
SMOVL C01013 +MOVJ EC01013
SMOVL C01014 +MOVJ EC01014
SMOVL C01015 +MOVJ EC01015
SMOVL C01016 +MOVJ EC01016
SMOVL C01017 +MOVJ EC01017
SMOVL C01018 +MOVJ EC01018
SMOVL C01019 +MOVJ EC01019
SMOVL C01020 +MOVJ EC01020
SMOVL C01021 +MOVJ EC01021
SMOVL C01022 +MOVJ EC01022
SMOVL C01023 +MOVJ EC01023
SMOVL C01024 +MOVJ EC01024
SMOVL C01025 +MOVJ EC01025
SMOVL C01026 +MOVJ EC01026
SMOVL C01027 +MOVJ EC01027
SMOVL C01028 +MOVJ EC01028
SMOVL C01029 +MOVJ EC01029
SMOVL C01030 +MOVJ EC01030
SMOVL C01031 +MOVJ EC01031
SMOVL C01032 +MOVJ EC01032
SMOVL C01033 +MOVJ EC01033
SMOVL C01034 +MOVJ EC01034
SMOVL C01035 +MOVJ EC01035
SMOVL C01036 +MOVJ EC01036
SMOVL C01037 +MOVJ EC01037
SMOVL C01038 +MOVJ EC01038
SMOVL C01039 +MOVJ EC01039
SMOVL C01040 +MOVJ EC01040
SMOVL C01041 +MOVJ EC01041
SMOVL C01042 +MOVJ EC01042
SMOVL C01043 +MOVJ EC01043
SMOVL C01044 +MOVJ EC01044
SMOVL C01045 +MOVJ EC01045
SMOVL C01046 +MOVJ EC01046
SMOVL C01047 +MOVJ EC01047
SMOVL C01048 +MOVJ EC01048
SMOVL C01049 +MOVJ EC01049
SMOVL C01050 +MOVJ EC01050
SMOVL C01051 +MOVJ EC01051
SMOVL C01052 +MOVJ EC01052
SMOVL C01053 +MOVJ EC01053
SMOVL C01054 +MOVJ EC01054
SMOVL C01055 +MOVJ EC01055
SMOVL C01056 +MOVJ EC01056
SMOVL C01057 +MOVJ EC01057
SMOVL C01058 +MOVJ EC01058
SMOVL C01059 +MOVJ EC01059
SMOVL C01060 +MOVJ EC01060
SMOVL C01061 +MOVJ EC01061
SMOVL C01062 +MOVJ EC01062
SMOVL C01063 +MOVJ EC01063
SMOVL C01064 +MOVJ EC01064
SMOVL C01065 +MOVJ EC01065
SMOVL C01066 +MOVJ EC01066
SMOVL C01067 +MOVJ EC01067
SMOVL C01068 +MOVJ EC01068
SMOVL C01069 +MOVJ EC01069
SMOVL C01070 +MOVJ EC01070
SMOVL C01071 +MOVJ EC01071
SMOVL C01072 +MOVJ EC01072
SMOVL C01073 +MOVJ EC01073
SMOVL C01074 +MOVJ EC01074
SMOVL C01075 +MOVJ EC01075
SMOVL C01076 +MOVJ EC01076
SMOVL C01077 +MOVJ EC01077
SMOVL C01078 +MOVJ EC01078
SMOVL C01079 +MOVJ EC01079
SMOVL C01080 +MOVJ EC01080
SMOVL C01081 +MOVJ EC01081
SMOVL C01082 +MOVJ EC01082
SMOVL C01083 +MOVJ EC01083
SMOVL C01084 +MOVJ EC01084
SMOVL C01085 +MOVJ EC01085
SMOVL C01086 +MOVJ EC01086
SMOVL C01087 +MOVJ EC01087
SMOVL C01088 +MOVJ EC01088
SMOVL C01089 +MOVJ EC01089
SMOVL C01090 +MOVJ EC01090
SMOVL C01091 +MOVJ EC01091
SMOVL C01092 +MOVJ EC01092
SMOVL C01093 +MOVJ EC01093
SMOVL C01094 +MOVJ EC01094
SMOVL C01095 +MOVJ EC01095
SMOVL C01096 +MOVJ EC01096
SMOVL C01097 +MOVJ EC01097
SMOVL C01098 +MOVJ EC01098
SMOVL C01099 +MOVJ EC01099
SMOVL C01100 +MOVJ EC01100
SMOVL C01101 +MOVJ EC01101
SMOVL C01102 +MOVJ EC01102
SMOVL C01103 +MOVJ EC01103
SMOVL C01104 +MOVJ EC01104
SMOVL C01105 +MOVJ EC01105
SMOVL C01106 +MOVJ EC01106
SMOVL C01107 +MOVJ EC01107
SMOVL C01108 +MOVJ EC01108
SMOVL C01109 +MOVJ EC01109
SMOVL C01110 +MOVJ EC01110
SMOVL C01111 +MOVJ EC01111
SMOVL C01112 +MOVJ EC01112
SMOVL C01113 +MOVJ EC01113
SMOVL C01114 +MOVJ EC01114
SMOVL C01115 +MOVJ EC01115
SMOVL C01116 +MOVJ EC01116
SMOVL C01117 +MOVJ EC01117
SMOVL C01118 +MOVJ EC01118
SMOVL C01119 +MOVJ EC01119
SMOVL C01120 +MOVJ EC01120
SMOVL C01121 +MOVJ EC01121
SMOVL C01122 +MOVJ EC01122
SMOVL C01123 +MOVJ EC01123
SMOVL C01124 +MOVJ EC01124
SMOVL C01125 +MOVJ EC01125
SMOVL C01126 +MOVJ EC01126
SMOVL C01127 +MOVJ EC01127
SMOVL C01128 +MOVJ EC01128
SMOVL C01129 +MOVJ EC01129
SMOVL C01130 +MOVJ EC01130
SMOVL C01131 +MOVJ EC01131
SMOVL C01132 +MOVJ EC01132
SMOVL C01133 +MOVJ EC01133
SMOVL C01134 +MOVJ EC01134
SMOVL C01135 +MOVJ EC01135
SMOVL C01136 +MOVJ EC01136
SMOVL C01137 +MOVJ EC01137
SMOVL C01138 +MOVJ EC01138
SMOVL C01139 +MOVJ EC01139
SMOVL C01140 +MOVJ EC01140
SMOVL C01141 +MOVJ EC01141
SMOVL C01142 +MOVJ EC01142
SMOVL C01143 +MOVJ EC01143
SMOVL C01144 +MOVJ EC01144
SMOVL C01145 +MOVJ EC01145
SMOVL C01146 +MOVJ EC01146
SMOVL C01147 +MOVJ EC01147
SMOVL C01148 +MOVJ EC01148
SMOVL C01149 +MOVJ EC01149
SMOVL C01150 +MOVJ EC01150
SMOVL C01151 +MOVJ EC01151
SMOVL C01152 +MOVJ EC01152
SMOVL C01153 +MOVJ EC01153
SMOVL C01154 +MOVJ EC01154
SMOVL C01155 +MOVJ EC01155
SMOVL C01156 +MOVJ EC01156
SMOVL C01157 +MOVJ EC01157
SMOVL C01158 +MOVJ EC01158
SMOVL C01159 +MOVJ EC01159
SMOVL C01160 +MOVJ EC01160
SMOVL C01161 +MOVJ EC01161
SMOVL C01162 +MOVJ EC01162
SMOVL C01163 +MOVJ EC01163
SMOVL C01164 +MOVJ EC01164
SMOVL C01165 +MOVJ EC01165
SMOVL C01166 +MOVJ EC01166
SMOVL C01167 +MOVJ EC01167
SMOVL C01168 +MOVJ EC01168
SMOVL C01169 +MOVJ EC01169
SMOVL C01170 +MOVJ EC01170
SMOVL C01171 +MOVJ EC01171
SMOVL C01172 +MOVJ EC01172
SMOVL C01173 +MOVJ EC01173
SMOVL C01174 +MOVJ EC01174
SMOVL C01175 +MOVJ EC01175
SMOVL C01176 +MOVJ EC01176
SMOVL C01177 +MOVJ EC01177
SMOVL C01178 +MOVJ EC01178
SMOVL C01179 +MOVJ EC01179
SMOVL C01180 +MOVJ EC01180
SMOVL C01181 +MOVJ EC01181
SMOVL C01182 +MOVJ EC01182
SMOVL C01183 +MOVJ EC01183
SMOVL C01184 +MOVJ EC01184
SMOVL C01185 +MOVJ EC01185
SMOVL C01186 +MOVJ EC01186
SMOVL C01187 +MOVJ EC01187
SMOVL C01188 +MOVJ EC01188
SMOVL C01189 +MOVJ EC01189
